// TIA Portal project "Tripping_hoya" (V16)

(* hardware
DEVICE "S7-1200 station_1"  S7-1200 Station
   slot 0: "Rack_0"  S7-1200 Rack  Rack  V1.0
   slot 1: "PLC_1"  CPU 1214C AC/DC/Rly  6ES7 214-1BG40-0XB0  V4.4
   slot 2: "DI 16x24VDC/DQ 16xRelay_1"  SM 1223 DI16/DQ16 x relay  6ES7 223-1PL32-0XB0  V2.0
   slot 3: "DI 16x24VDC/DQ 16xRelay_2"  SM 1223 DI16/DQ16 x relay  6ES7 223-1PL32-0XB0  V2.0
   slot 4: "DI 16x24VDC/DQ 16xRelay_3"  SM 1223 DI16/DQ16 x relay  6ES7 223-1PL32-0XB0  V2.0
   slot 5: "DQ 8x24VDC _1"  SM 1222 DQ8 x 24VDC  6ES7 222-1BF32-0XB0  V2.0
   slot 6: "DI 16x24VDC_1"  6ES7 221-1BH32-0XB0  V2.0
   slot 7: "DI 16x24VDC_2"  6ES7 221-1BH32-0XB0  V2.0
   slot 101: "CM 1241 (RS232)_1"  6ES7 241-1AH32-0XB0  V2.2
*)

// ===== PLC "PLC_1"  CPU 1214C AC/DC/Rly =====

VAR_GLOBAL   // PLC tag table "Default tag table"
   "Start" AT %I0.0 : Bool;   // Tín hiệu nhấn nút start
   "Stop" AT %I0.1 : Bool;   // Tín hiệu nhấn nút stop
   "Reset" AT %I0.2 : Bool;   // Tín hiệu nhấn nút Reset
   "EMG" AT %I0.3 : Bool;
   "SS Up XL Chốt" AT %I0.4 : Bool;
   "SS Down XL Chốt" AT %I0.5 : Bool;
   "SS Up XL Cửa Input" AT %I0.6 : Bool;
   "SS Down XL Cửa Input" AT %I0.7 : Bool;
   "SS Up XL Nâng Input" AT %I1.0 : Bool;
   "SS Down XL Nâng Input" AT %I1.1 : Bool;
   "SS Input Rack" AT %I1.2 : Bool;   // Cảm biến có rack trong Xylanh nâng input
   "SS Chốt Rack Input" AT %I1.3 : Bool;
   "SS Rack Input XL" AT %I1.4 : Bool;
   "SS Limit 1 Tranfer1" AT %I1.5 : Bool;
   "SS Limit 1 Tranfer2" AT %I2.1 : Bool;
   "SS Open XL Robot" AT %I2.3 : Bool;
   "SS Close XL Robot" AT %I2.4 : Bool;
   "SS Down XL Robot" AT %I2.5 : Bool;
   "SS Up XL Robot" AT %I2.6 : Bool;   // Cảm biến Xy Lanh dọc của Robot
   "SS XL Up Cửa Output" AT %I2.7 : Bool;
   "SS XL Down Cửa Output" AT %I3.0 : Bool;
   "SS Up XL Nâng Output" AT %I3.1 : Bool;
   "SS Down XL Nâng Output" AT %I3.2 : Bool;
   "SS Up XL Lift 1" AT %I5.5 : Bool;
   "SS Down XL Lift 1" AT %I5.6 : Bool;   // Trgger DOwnnXLn3
   "SS Up XL Lift 5" AT %I5.7 : Bool;
   "SS Down XL Lift 5" AT %I6.0 : Bool;
   "SS HW Tank1" AT %I6.1 : Bool;
   "SS LW Tank1" AT %I6.2 : Bool;
   "SS HW Tank2" AT %I6.3 : Bool;
   "SS LW Tank2" AT %I6.4 : Bool;
   "SS HW Tank3" AT %I6.5 : Bool;
   "SS LW Tank3" AT %I6.6 : Bool;
   "SS HW Tank4" AT %I6.7 : Bool;
   "SS LW Tank4" AT %I7.0 : Bool;
   "SS HW Tank5" AT %I7.1 : Bool;
   "SS LW Tank5" AT %I7.2 : Bool;
   "SS HW Tank6" AT %I7.3 : Bool;
   "SS LW Tank6" AT %I7.4 : Bool;
   "SS HW Tank7" AT %I7.5 : Bool;
   "SS LW Tank7" AT %I7.6 : Bool;
   "SS HW Tank8" AT %I7.7 : Bool;
   "SS LW Tank8" AT %I8.0 : Bool;
   "SS HW Tank9" AT %I8.1 : Bool;
   "SS LW Tank9" AT %I8.2 : Bool;
   "SS W Tank1" AT %I8.5 : Bool;
   "SS W Tank2" AT %I8.6 : Bool;
   "SS W Tank3" AT %I8.7 : Bool;
   "SS W Tank4" AT %I9.0 : Bool;
   "SS W Tank5" AT %I9.1 : Bool;
   "SS W Tank6" AT %I9.2 : Bool;
   "SS W Tank7" AT %I9.3 : Bool;
   "SS W Tank8" AT %I9.4 : Bool;
   "SS W Tank9" AT %I9.5 : Bool;
   "SS Rack BT Out" AT %I9.7 : Bool;
   "Up_Limit_Lift" AT %I10.2 : Bool;   // Cảm Biến Trên Axis Lift
   "Down_Limit_Lift" AT %I10.3 : Bool;   // Cảm biến Dưới Axis Lift
   "Jog + Robot" AT %I10.4 : Bool;   // Trigger JOG +
   "Jog - Robot" AT %I10.5 : Bool;   // Trigger JOG -
   "SS Up XL Lift 2" AT %I10.6 : Bool;   // Cảm Biến Trên Xy Lanh Nâng Bath 4
   "SS Down XL Lift 2" AT %I10.7 : Bool;   // Cảm Biến Dưới Xy Lanh Nâng Bath 4
   "SS Up XL Lift 3" AT %I11.0 : Bool;   // Cảm Biến Trên Xy Lanh Nâng Bath 5
   "SS Down XL Lift 3" AT %I11.1 : Bool;   // Cảm Biến Dưới Xy Lanh Nâng Bath 5
   "SS Up XL Lift 4" AT %I11.2 : Bool;   // Cảm Biến Trên Xy Lanh Nâng Bath 6
   "SS Down XL Lift 4" AT %I11.3 : Bool;   // Cảm Biến Dưới Xy Lanh Nâng Bath 6
   "SS_Cửa_Khung" AT %I11.4 : Bool;
   "Right_Limit_X" AT %I11.5 : Bool;
   "Left_Limit_X" AT %I11.6 : Bool;
   "XL Chốt Input_1" AT %Q0.0 : Bool;
   "XL Chốt Input_2" AT %Q0.1 : Bool;
   "XL Cửa Input_1" AT %Q0.2 : Bool;
   "XL Cửa Input_2" AT %Q0.3 : Bool;
   "XL Nâng Input1" AT %Q0.4 : Bool;
   "XL Nâng Input2" AT %Q0.5 : Bool;
   "XL Kẹp Robot_1" AT %Q0.6 : Bool;
   "XL Kẹp Robot_2" AT %Q0.7 : Bool;
   "Motor Băng tải Input" AT %Q1.0 : Bool;
   "XL Cửa Output_1" AT %Q1.1 : Bool;
   "XL Cửa Output_2" AT %Q2.0 : Bool;
   "XL Nâng Output1" AT %Q2.1 : Bool;
   "XL Nâng Output2" AT %Q2.2 : Bool;
   "Motor Băng Tải Output" AT %Q2.3 : Bool;
   "Van DI ON" AT %Q2.4 : Bool;
   "Van DI OFF" AT %Q2.5 : Bool;
   "Pump Bath1" AT %Q2.6 : Bool;
   "Pump Bath2" AT %Q2.7 : Bool;
   "Pump Bath3" AT %Q3.0 : Bool;
   "Pump Bath4" AT %Q3.1 : Bool;
   "Pump Bath5" AT %Q3.2 : Bool;
   "Pump Bath6" AT %Q3.3 : Bool;
   "Pump Bath7" AT %Q3.4 : Bool;
   "Pump Bath8" AT %Q3.5 : Bool;
   "Pump Bath9" AT %Q3.6 : Bool;
   "Pump Bath10" AT %Q3.7 : Bool;
   "Van RO ON" AT %Q4.0 : Bool;
   "Van RO OFF" AT %Q4.1 : Bool;
   "UltraS Tank1" AT %Q4.5 : Bool;
   "UltraS Tank2" AT %Q4.6 : Bool;
   "UltraS Tank3" AT %Q4.7 : Bool;
   "UltraS Tank4" AT %Q5.0 : Bool;
   "UltraS Tank5" AT %Q5.1 : Bool;
   "UltraS Tank6" AT %Q5.2 : Bool;
   "UltraS Tank7" AT %Q5.3 : Bool;
   "UltraS Tank8" AT %Q5.4 : Bool;
   "UltraS Tank9" AT %Q5.5 : Bool;
   "XL Lift 1_1" AT %Q6.0 : Bool;
   "XL Lift 1_2" AT %Q6.1 : Bool;
   "XL Lift 2_1" AT %Q6.2 : Bool;
   "XL Lift 2_2" AT %Q6.3 : Bool;
   "XL Lift 3_1" AT %Q6.4 : Bool;
   "XL Lift 3_2" AT %Q6.5 : Bool;
   "XL Lift 4_1" AT %Q6.6 : Bool;
   "XL Lift 4_2" AT %Q6.7 : Bool;
   "XL Lift 5_1" AT %Q7.0 : Bool;
   "XL Lift 5_2" AT %Q7.1 : Bool;
   "Red Lamp" AT %Q7.2 : Bool;
   "Yellow Lamp" AT %Q7.3 : Bool;
   "Green Lamp" AT %Q7.4 : Bool;
   "Buzzer" AT %Q7.5 : Bool;
   "XL_UP_Robot" AT %Q7.6 : Bool;
   "XL_DOWN_Robot" AT %Q7.7 : Bool;
   "System_Byte" AT %MB1 : Byte;
   "FirstScan" AT %M1.0 : Bool;
   "DiagStatusUpdate" AT %M1.1 : Bool;
   "AlwaysTRUE" AT %M1.2 : Bool;
   "AlwaysFALSE" AT %M1.3 : Bool;
   "Clock_Byte" AT %MB0 : Byte;
   "Clock_10Hz" AT %M0.0 : Bool;
   "Clock_5Hz" AT %M0.1 : Bool;
   "Clock_2.5Hz" AT %M0.2 : Bool;
   "Clock_2Hz" AT %M0.3 : Bool;
   "Clock_1.25Hz" AT %M0.4 : Bool;
   "Clock_1Hz" AT %M0.5 : Bool;
   "Clock_0.625Hz" AT %M0.6 : Bool;
   "Clock_0.5Hz" AT %M0.7 : Bool;
   "DISCONNECT_TCP_PC_TRGGER" AT %M2.0 : Bool;   // Tín hiệu ngắt kết nối từ PC
   "SEND_TCP_TRIGGER" AT %M2.1 : Bool;   // Tín Hiệu Gửi TCP 1
   "SEND_TCP_TRIGGER_1" AT %M2.2 : Bool;   // Tín Hiệu Gủi TCP 2
   "SEND_TCP_TRIGGER_2" AT %M2.3 : Bool;   // Tín Hiệu Gửi TCP 3
   "SEND_REQ" AT %M2.4 : Bool;   // Tín Hiệu Kích Gửi
   "length" AT %MW4 : Int;   // Biến Lưu Chiều Dài Data cần gửi
   "Edge_1" AT %M2.5 : Bool;   // Temp Pulse 1
   "Axis_x_Home" AT %M2.6 : Bool;   // Axis X Home trigger
   "Edge_2" AT %M2.7 : Bool;   // Temp Pulse 2
   "SYSTEM_READY" AT %M3.0 : Bool;   // READY STATUS
   "MANUAL_STATE" AT %M3.1 : Bool;   // Chế độ manual
   "AUTO_STATE" AT %M3.2 : Bool;   // Chế Dộ AUTO
   "HOME_MAN_TRIGGER_PC" AT %M3.3 : Bool;   // Tín Hiệu Home Manual
   "HOME_AUTO_TRIGGER_PC" AT %M3.4 : Bool;   // Tín HIệu HOME AUTO
   "SELECT_AXIS_HOME" AT %MW6 : Int;   // 0-ALL Axis , 1 - AXIS X, 2 - AXIS LIFT
   "Edge_3" AT %M3.5 : Bool;   // Temp Pulse 3
   "Edge_4" AT %M3.6 : Bool;   // Temp Pulse 4
   "Edge_5" AT %M3.7 : Bool;   // Temp 5
   "Edge_6" AT %M8.0 : Bool;   // Temp6
   "Edge_7" AT %M8.1 : Bool;   // Temp 7
   "Edge_8" AT %M8.2 : Bool;   // Temp 8
   "Edge_9" AT %M8.3 : Bool;   // Temp 9
   "Edge_10" AT %M8.4 : Bool;   // Temp 10
   "Move_Point_X" AT %M8.5 : Bool;   // Trigger_Move_Point Axis X
   "Edge_11" AT %M8.6 : Bool;   // Temp 11
   "Move_Point_LIFT" AT %M8.7 : Bool;   // Tín Hiệu Move Point Axis LIFT
   "WRITE_DATA_POINT_X" AT %M9.0 : Bool;   // Trigger Cài đặt điểm
   "Edge_12" AT %M9.1 : Bool;   // Temp 12
   "Edge_13" AT %M9.2 : Bool;   // Temp 13
   "WRITE_DATA_POINT_LIFT" AT %M9.3 : Bool;   // Trigger Set data point Axis LIft
   "Jog_TF_1_FW" AT %M9.4 : Bool;   // Trigger Jog FW Tranfer 1
   "Edge_14" AT %M9.5 : Bool;   // Temp 14
   "Edge_15" AT %M9.6 : Bool;   // Temp 15
   "Edge_16" AT %M9.7 : Bool;   // Temp 16
   "Edge_17" AT %M10.0 : Bool;   // Temp 17
   "Jog_TF_1_BW" AT %M10.1 : Bool;   // Trigger Jog BW Tranfer 1
   "Jog_TF_2_FW" AT %M10.2 : Bool;   // Trigger Jog FW Tranfer 2
   "Edge_18" AT %M10.3 : Bool;   // Temp 18
   "Edge_19" AT %M10.4 : Bool;   // Temp 19
   "Jog_TF_2_BW" AT %M10.5 : Bool;   // Trigger Jog BW Tranfer 2
   "Edge_20" AT %M10.6 : Bool;   // Temp 20
   "Edge_21" AT %M10.7 : Bool;   // Temp 21
   "Run_TF_1_FW" AT %M11.0 : Bool;   // Trgger Run FW Tranfer 1
   "Edge_22" AT %M11.1 : Bool;   // Temp 22
   "Edge_23" AT %M11.2 : Bool;   // Temp 23
   "Run_TF_1_BW" AT %M11.3 : Bool;   // Trgger Run BW Tranfer 1
   "Edge_24" AT %M11.4 : Bool;   // Temp 24
   "Edge_25" AT %M11.5 : Bool;   // Temp 25
   "Run_TF_2_FW" AT %M11.6 : Bool;   // Trigger Run FW Tranfer 2
   "Edge_26" AT %M11.7 : Bool;   // Temp 26
   "Edge_27" AT %M12.0 : Bool;   // Temp 27
   "Run_TF_2_BW" AT %M12.1 : Bool;   // Trigger Run BW Tranfer 2
   "Edge_28" AT %M12.2 : Bool;   // Temp 28
   "Edge_29" AT %M12.3 : Bool;   // Temp 29
   "Jog_Lift_1_FW" AT %M12.4 : Bool;   // Trigger Jog Lift 1 FW
   "Edge_30" AT %M12.5 : Bool;   // Temp 30
   "Edge_31" AT %M12.6 : Bool;   // Temp 31
   "Jog_Lift_1_BW" AT %M12.7 : Bool;   // Trgger Jog Lift 1 BW
   "Edge_32" AT %M13.0 : Bool;   // Temp 32
   "Edge_33" AT %M13.1 : Bool;   // Temp 33
   "Run_Lift_1_FW" AT %M13.2 : Bool;   // Trigger Run Lift 1 FW
   "Edge_34" AT %M13.3 : Bool;   // Temp 34
   "Edge_35" AT %M13.4 : Bool;   // Temp 35
   "Run_Lift_1_BW" AT %M13.5 : Bool;   // Trigger Run Lift 1 BW
   "Edge_36" AT %M13.6 : Bool;   // Temp 36
   "Edge_37" AT %M13.7 : Bool;   // Temp 37
   "Jog_Lift_2_FW" AT %M14.0 : Bool;   // Trigger Jog Lifft 2 FW
   "Edge_38" AT %M14.1 : Bool;   // Temp 38
   "Edge_39" AT %M14.2 : Bool;   // Temp 39
   "Jog_Lift_2_BW" AT %M14.3 : Bool;   // Trigger Jog Lift 2 BW
   "Edge_40" AT %M14.4 : Bool;   // Temp 40
   "Edge_41" AT %M14.5 : Bool;   // Temp 41
   "Run_Lift_2_FW" AT %M14.6 : Bool;   // Trigger Run Lift 2 FW
   "Edge_42" AT %M14.7 : Bool;   // Temp 42
   "Edge_43" AT %M15.0 : Bool;   // Temp 43
   "Run_Lift_2_BW" AT %M15.1 : Bool;   // Trigger Run Lifr 2 BW
   "Edge_44" AT %M15.2 : Bool;   // Temp 44
   "Edge_45" AT %M15.3 : Bool;   // Temp 45
   "Jog_Lift_3_FW" AT %M15.4 : Bool;   // Trgger Jog Lift 3 FW
   "Edge_46" AT %M15.5 : Bool;   // Temp 46
   "Edge_47" AT %M15.6 : Bool;   // Temp 47
   "Jog_Lift_3_BW" AT %M15.7 : Bool;   // Trigger Jog Lift 3 BW
   "Edge_48" AT %M16.0 : Bool;   // Temp 48
   "Edge_49" AT %M16.1 : Bool;   // Temp 49
   "Run_Lift_3_FW" AT %M16.2 : Bool;   // Trigger Run Lift 3 FW
   "Edge_50" AT %M16.3 : Bool;   // Temp 50
   "Edge_51" AT %M16.4 : Bool;   // Temp 51
   "Run_Lift_3_BW" AT %M16.5 : Bool;   // Trigger Run Lift 3 BW
   "Edge_52" AT %M16.6 : Bool;   // Temp 52
   "Edge_53" AT %M16.7 : Bool;   // Temp 53
   "SET_FREQ_MOTOR_TRANFER" AT %M17.0 : Bool;   // Tín hiệu set freq cho Motor tranfer
   "SET_ACC_DEC_MOTOR_TRANFER" AT %M17.1 : Bool;
   "Edge_54" AT %M17.2 : Bool;   // Temp 54
   "Edge_55" AT %M17.3 : Bool;   // Temp 55
   "SET_FREQ_MOTOR_LIFT" AT %M17.4 : Bool;   // Tín hiệu cài đặt tần số cho đọng cơ nhúng
   "Edge_56" AT %M17.5 : Bool;   // Temp 56
   "SET_ACC_DEC_MOTOR_LIFT" AT %M17.6 : Bool;   // Tín hiệu cài đặt thời gian tăng tốc giảm tốc của động cơ nhúng
   "Edge_57" AT %M17.7 : Bool;   // Temp 57
   "Man_Axis_X" AT %I8.3 : Bool;   // Biến Chọn Manual Axis X
   "Man_Axis_Lift" AT %I8.4 : Bool;   // Biến Chọn Manual Axis Lift
   "Begin_Reset" AT %M18.0 : Bool;   // Reset Trgger
   "Stop_Pump_temp_1" AT %M18.1 : Bool;
   "RESET_PUMP_1" AT %M18.2 : Bool;
   "START_PUMP_1" AT %M18.3 : Bool;
   "STOP_PUMP_1" AT %M18.4 : Bool;
   "Stop_Pump_temp_2" AT %M18.5 : Bool;
   "RESET_PUMP_2" AT %M18.6 : Bool;
   "START_PUMP_2" AT %M18.7 : Bool;
   "STOP_PUMP_2" AT %M19.0 : Bool;
   "Stop_Pump_temp_3" AT %M19.1 : Bool;
   "RESET_PUMP_3" AT %M19.2 : Bool;
   "START_PUMP_3" AT %M19.3 : Bool;
   "STOP_PUMP_3" AT %M19.4 : Bool;
   "Stop_Pump_temp_4" AT %M19.5 : Bool;
   "RESET_PUMP_4" AT %M19.6 : Bool;
   "START_PUMP_4" AT %M19.7 : Bool;
   "STOP_PUMP_4" AT %M20.0 : Bool;
   "Stop_Pump_temp_5" AT %M20.1 : Bool;
   "RESET_PUMP_5" AT %M20.2 : Bool;
   "START_PUMP_5" AT %M20.3 : Bool;
   "STOP_PUMP_5" AT %M20.4 : Bool;
   "Stop_Pump_temp_6" AT %M20.5 : Bool;
   "RESET_PUMP_6" AT %M20.6 : Bool;
   "START_PUMP_6" AT %M20.7 : Bool;
   "STOP_PUMP_6" AT %M21.0 : Bool;
   "Stop_Pump_temp_7" AT %M21.1 : Bool;
   "RESET_PUMP_7" AT %M21.2 : Bool;
   "START_PUMP_7" AT %M21.3 : Bool;
   "STOP_PUMP_7" AT %M21.4 : Bool;
   "Stop_Pump_temp_8" AT %M21.5 : Bool;
   "START_PUMP_8" AT %M21.6 : Bool;
   "RESET_PUMP_8" AT %M21.7 : Bool;
   "STOP_PUMP_8" AT %M22.0 : Bool;
   "Stop_Pump_temp_9" AT %M22.1 : Bool;
   "RESET_PUMP_9" AT %M22.2 : Bool;
   "STOP_PUMP_9" AT %M22.3 : Bool;
   "START_PUMP_9" AT %M22.4 : Bool;
   "Home_Tranfer" AT %M22.5 : Bool;   // Home Tranfer
   "Edge_58" AT %M22.6 : Bool;   // Temp 58
   "Initial_Tranfer" AT %M22.7 : Bool;   // Initail Tranfer Group
   "Stop_JOG_Tranfer" AT %M23.0 : Bool;   // Stop Signal Tranfer
   "Current_timer_Count" AT %MD24 : Time;   // Biến nhớ Time Hiện Tại
   "Prepare_BW_TF_1" AT %M23.1 : Bool;   // Signal backward tranfer group
   "Edge_59" AT %M23.2 : Bool;   // Temp 59
   "Edge_60" AT %M23.3 : Bool;   // Temp 60
   "BW_Tranfer" AT %M23.4 : Bool;   // Signal Trigger BW
   "Edge_61" AT %M23.5 : Bool;   // Temp 61
   "Up_XL_Lift_1" AT %M23.6 : Bool;   // Trigger Up Xy Lanh 1
   "Down_XL_Lift_1" AT %M23.7 : Bool;   // Trigger Down Xy Lạnh 1
   "Down_XL_Lift_2" AT %M28.0 : Bool;   // Trgger Down XL 2
   "Up_XL_Lift_2" AT %M28.1 : Bool;   // Trigger Up XL 2
   "Up_XL_Lift_3" AT %M28.2 : Bool;   // Trigger XL Lift 3
   "Down_XL_Lift_3" AT %M28.3 : Bool;   // Trigger Down XL Lift 3
   "Up_XL_Lift_4" AT %M28.4 : Bool;   // Trgger Up XL Lift 4
   "Down_XL_Lift_4" AT %M28.5 : Bool;   // Trgger Down XL Lift 4
   "Up_XL_Lift_5" AT %M28.6 : Bool;   // Trgger Up XL Lift 5
   "Down_XL_Lift_5" AT %M28.7 : Bool;   // Trigger Down XL 5
   "Manual_Up_XL_Lift_1" AT %M29.0 : Bool;   // Trigger Manual Up XL Lift 1
   "Manual_Down_XL_Lift_1" AT %M29.1 : Bool;   // Trigger manual Down XL Lift 1
   "Manual_Up_XL_Lift_2" AT %M29.2 : Bool;   // Trgger Manual Up XL Lift 2
   "Manual_Down_XL_Lift_2" AT %M29.3 : Bool;   // Trigger Manual Down XL Lift 2
   "Manual_Up_XL_Lift_3" AT %M29.4 : Bool;   // Trigger Manual Up XL Lift 3
   "Manual_Down_XL_Lift_3" AT %M29.5 : Bool;   // Trigger Manual Down XL Lift 3
   "Manual_Up_XL_Lift_4" AT %M29.6 : Bool;   // Trigger Manual Up XL Lift 4
   "Manual_Down_XL_Lift_4" AT %M29.7 : Bool;   // Trigger Manual Down XL Lift 4
   "Manual_Up_XL_Lift_5" AT %M30.0 : Bool;   // Trigger Manual Up XL Lift 5
   "Manual_Down_XL_Lift_5" AT %M30.1 : Bool;   // Trigger Manual Down XL Lift 5
   "Up_XL_Chốt" AT %M30.2 : Bool;   // Signal Up Xy Lanh Chốt
   "Manual_Up_XL_Chốt_Input" AT %M30.3 : Bool;   // Trigger manual Up Xy Lanh Chốt In put
   "Down_XL_Chốt" AT %M30.4 : Bool;   // Trigger Down Xy Lanh Chốt Input
   "Manual_Down_XL_Chốt_Input" AT %M30.5 : Bool;   // Trigger Manual Down Xy lanh CHót Input
   "Up_XL_Nâng Input" AT %M30.6 : Bool;   // Trigger Up XL nâng input
   "Manual_Up_XL_Nâng_Input" AT %M30.7 : Bool;   // Trigger manual up Xy lanh nâng input
   "Down_XL_Nâng Input" AT %M31.0 : Bool;   // Trigger Down XL Nâng input
   "Manual_Down_XL_Nâng_Input" AT %M31.1 : Bool;   // Trigger Manual Down XL nâng input
   "Up_XL_Nâng Output" AT %M31.2 : Bool;   // Trigger Up XL Nâng Input
   "Down_XL_Nâng Output" AT %M31.3 : Bool;   // Trigger Up XL Nâng Output
   "Manual_Down_XL_Nâng_ Output" AT %M31.4 : Bool;   // Trigger Manual Down XL Nâng Input
   "CLose_XL_Kẹp_Robot" AT %M31.5 : Bool;   // Trigger Close XL Kẹp Robot
   "Manual_Close_XL_Kẹp_Robot" AT %M31.6 : Bool;   // Trigger Manual Close Xl Kẹp Robot
   "Open_XL_Kẹp_Robot" AT %M31.7 : Bool;   // Trigger Open XL Kẹp Robot
   "Manual_Open_XL_Kẹp_Robot" AT %M32.0 : Bool;   // Trigger Manual Open XL Kẹp Robot
   "Up_XL_Robot" AT %M32.1 : Bool;   // Trigger Up XL Robot
   "Manual_Up_XL_Robot" AT %M32.2 : Bool;   // Trigger Manual Up XL Robot
   "Down_XL_Robot" AT %M32.3 : Bool;   // Trigger Down XL Robot
   "Manual_Down_XL_Robot" AT %M32.4 : Bool;   // Trigger Manual Down XL Robot
   "Edge_62" AT %M32.5 : Bool;   // Temp 62
   "No_rack" AT %M32.6 : Bool;   // Signal Detect Has Any Rack In Machine
   "TF1_Position_1" AT %M32.7 : Bool;   // Signal Detect TF1 at Position 1
   "Trigger_Run_FW_TF1" AT %M33.0 : Bool;   // Signal Run FW TF Excute
   "TF1_Position_2" AT %M33.1 : Bool;   // Signal Detect Tranfer 1 at Position 2
   "Stop_Run_FW_TF1" AT %M33.2 : Bool;   // Signal to Stop Run Forward Tranffer 1
   "Stop_Run_BW_TF1" AT %M33.3 : Bool;   // Signal to stop run backward Tranfer 1
   "Trigger_Run_BW_TF1" AT %M33.4 : Bool;   // Signal Run Backward Tranfer1
   "Being_TF1_FW" AT %M33.5 : Bool;   // Status FW of TF1
   "Being_TF1_BW" AT %M33.6 : Bool;   // Status BW of TF1
   "Mem_Status_1" AT %M33.7 : Bool;   // Memory 1
   "Begin_Tripping" AT %M34.0 : Bool;   // Signal To Tripping Area 1
   "Edge_63" AT %M34.1 : Bool;   // Temp 63
   "Down_XL_Lift_1_Excute" AT %M34.2 : Bool;   // Excute Down XL Lift 1
   "Edge_64" AT %M34.3 : Bool;   // Temp 64
   "Stop_Delay_Temp_1" AT %M34.4 : Bool;   // Mem temp 1
   "Tripping_Area1_Done" AT %M34.5 : Bool;   // Signal Detect Tripping Process Done
   "Up_XL_Lift_1_Excute" AT %M34.6 : Bool;   // Excute Up XL Liff 1
   "Trigger_Trip_Area1" AT %M34.7 : Bool;   // Trigger To Excute Begin Tranffer
   "Trigger_Trip_Area3" AT %M35.0 : Bool;   // Trigger to Excute Tripping process Area 3
   "TF2_Position_1" AT %M35.1 : Bool;   // Signal Detect TF2 at Possiontion 1
   "TF2_Position_2" AT %M35.2 : Bool;   // Signal Detect TF2 at Position 2
   "Stop_Run_FW_TF2" AT %M35.3 : Bool;   // Stop Signal Run TF2 FW
   "Trigger_Run_FW_TF2" AT %M35.4 : Bool;   // Trigger to Run FW TF2
   "Being_TF2_FW" AT %M35.5 : Bool;   // Status Run FW TF2
   "Stop_Run_BW_TF2" AT %M35.6 : Bool;   // Signal To Stop Run BW TF2
   "Trigger_Run_BW_TF2" AT %M35.7 : Bool;   // Trigger to Run BW TF2
   "Being_TF2_BW" AT %M36.0 : Bool;   // Status Run BW TF2
   "Down_XL_Lift_5_Excute" AT %M36.1 : Bool;   // Trigger Down XL 5 Excute
   "Mem_Status_2" AT %M36.2 : Bool;   // Memory temp 2
   "Begin_Tripping_1" AT %M36.3 : Bool;   // Signal To Tripping Area3
   "Stop_Delay_Temp_2" AT %M36.4 : Bool;   // Mem Temp 2
   "Edge_65" AT %M36.5 : Bool;   // Temp 65
   "Edge_66" AT %M36.6 : Bool;   // Temp 66
   "Up_XL_Lift_5_Excute" AT %M36.7 : Bool;   // Excute Up XL Lift 5
   "Back_To_Posiont1_TF1" AT %M37.0 : Bool;   // Signal to back to postion 1
   "Prepare_Stop_TF1" AT %M37.1 : Bool;   // Signal To prepare stop TF1
   "Descrease_Speed_TF1" AT %M37.2 : Bool;   // Signal To Descrease Speed Of Tranfer 1
   "Edge_67" AT %M37.3 : Bool;   // Temp 67
   "Edge_68" AT %M37.4 : Bool;   // Temp 68
   "Waiting_SS_off_1" AT %M37.5 : Bool;   // Biến đợi cảm biến tắt lần 1
   "Edge_69" AT %M37.6 : Bool;   // Temp 69
   "Jog_home_TF1_BW_Excute" AT %M37.7 : Bool;   // Trigger Jog BW TF1 (1)
   "Waiting_SS_on_1" AT %M38.0 : Bool;   // Biến Đợi Cảm Biến TF1 On
   "Edge_70" AT %M38.1 : Bool;   // Temp70
   "Edge_71" AT %M38.3 : Bool;   // Temp 71
   "Original_TF" AT %M38.4 : Bool;   // ON: Đã Về gốc Tranfer, OFF: Đang hoặc chưa được về gốc
   "Edge_72" AT %M38.5 : Bool;   // Temp 72
   "Edge_73" AT %M38.6 : Bool;   // Temp 73
   "Edge_74" AT %M38.7 : Bool;   // Temp 74
   "Stop_JOG_Tranfer_1" AT %M39.0 : Bool;
   "Back_To_Posiont1_TF2" AT %M39.1 : Bool;
   "Original_TF_2" AT %M39.2 : Bool;
   "Prepare_Stop_TF2" AT %M39.3 : Bool;
   "Edge_75" AT %M39.4 : Bool;   // Temp 75
   "Edge_76" AT %M39.5 : Bool;   // Temp 76
   "Jog_home_TF2_BW_Excute" AT %M39.6 : Bool;
   "Current_timer_Count_2" AT %MD40 : Time;
   "Prepare_BW_TF_2" AT %M39.7 : Bool;
   "Initial_Tranfer_2" AT %M44.0 : Bool;
   "Waiting_SS_off_3" AT %M44.1 : Bool;
   "Edge_77" AT %M44.2 : Bool;
   "Edge_78" AT %M44.3 : Bool;
   "Waiting_SS_on_3" AT %M44.4 : Bool;
   "Prepare_BW_TF_3" AT %M44.5 : Bool;
   "Edge_79" AT %M44.6 : Bool;
   "Waiting_SS_off_4" AT %M44.7 : Bool;
   "Edge_80" AT %M45.0 : Bool;
   "Tripping_Area3_Done" AT %M45.1 : Bool;
   "Move_Avoid" AT %M45.2 : Bool;   // Trigger move to avoid robot
   "Move_Avoid_Excute" AT %M45.3 : Bool;   // Biến thực thi tránh robot
   "Stop_Move_Avoid" AT %M45.4 : Bool;   // Trigger To stop Avoid
   "Move_back_after_avoid" AT %M45.5 : Bool;
   "Move_back_after_avoid_Excute" AT %M45.6 : Bool;
   "Stop_Move_Back_Avoid" AT %M45.7 : Bool;
   "Signal_Active_Robot" AT %M46.0 : Bool;   // Tín hiệu báo hiệu khỏi động robot cho quá trình vove rack
   "Edge_81" AT %M46.1 : Bool;   // Temp 81
   "Start_Grab_Robot" AT %M46.2 : Bool;
   "Pick_From4_to_6" AT %M46.3 : Bool;   // Tín hiều di chuyển Rack từ Bath 4 đến Bath6
   "Pick_From4_to_5" AT %M46.4 : Bool;   // Tin hiệu di chuyển Rack dến Bath 5
   "At_Bath4" AT %M46.5 : Bool;   // Tín hiệu CHo biết Rack sẽ được nhúng ở Bath 4
   "Re_Signal_Start_Grab_Robot" AT %M46.6 : Bool;   // Tín hiệu gọi lại CỤm Robot
   "Move_Preocess_Robot_Excute" AT %M46.7 : Bool;   // Biến Khởi Động Chu trình Robot
   "Edge_82" AT %M47.0 : Bool;   // Temp 82
   "Robot_Move_P1_Started" AT %M47.1 : Bool;
   "Grabed_Rack" AT %M47.2 : Bool;   // Tín Hiệu báo hiệu đã kẹp rack
   "Pick_P1_Done" AT %M47.3 : Bool;   // Pick At P1 Robot Done
   "Edge_83" AT %M47.4 : Bool;   // Temp 83
   "Robot_Move_P2_Started" AT %M47.5 : Bool;
   "Edge_84" AT %M47.6 : Bool;   // Temp 84
   "Down_XL_Robot_1" AT %M47.7 : Bool;
   "Open_XL_Kẹp_Robot_1" AT %M48.0 : Bool;
   "Put_Rack_to_Bath" AT %M48.1 : Bool;
   "Up_XL_Robot_1" AT %M48.2 : Bool;
   "Put_Rack_Done" AT %M48.3 : Bool;
   "Edge_85" AT %M48.4 : Bool;   // Temp 85
   "Down_XL_Lift_Trgger" AT %M48.5 : Bool;
   "Down_XL_Lift_2_1" AT %M48.6 : Bool;
   "Down_XL_Lift_3_1" AT %M48.7 : Bool;
   "Down_XL_Lift_4_1" AT %M49.0 : Bool;
   "Manual_Jog + Robot" AT %M49.1 : Bool;   // Biến Manual Jog
   "Manual_Jog - Robot" AT %M49.2 : Bool;
   "Axis_X_Selection" AT %I3.3 : Bool;
   "Axis_Lift_Selection" AT %I3.4 : Bool;
   "Manual_Jog + Lift" AT %M49.3 : Bool;
   "Manual_Jog - Lift" AT %M49.4 : Bool;
   "Enable_Robot" AT %M49.5 : Bool;
   "Edge_86" AT %M49.6 : Bool;   // Temp 86
   "Disable_Robot" AT %M49.7 : Bool;
   "Edge_87" AT %M50.0 : Bool;   // Temp87
   "Enable_Lift" AT %M50.1 : Bool;
   "Edge_88" AT %M50.2 : Bool;   // Temp 88
   "Disable_Lift" AT %M50.3 : Bool;
   "Edge_89" AT %M50.4 : Bool;   // Temp 89
   "Manual_Jog_FW_TF1" AT %M50.5 : Bool;
   "Edge_90" AT %M50.6 : Bool;   // Temp 90
   "Edge_91" AT %M50.7 : Bool;   // Temp 91
   "Manual_Jog_BW_TF1" AT %M51.0 : Bool;
   "Edge_92" AT %M51.1 : Bool;
   "Edge_93" AT %M51.2 : Bool;
   "Manual_Jog_FW_TF2" AT %M51.3 : Bool;
   "Manual_Jog_BW_TF2" AT %M51.4 : Bool;
   "Edge_94" AT %M51.5 : Bool;   // Temp 94
   "Edge_95" AT %M51.6 : Bool;   // Temp96
   "Edge_96" AT %M51.7 : Bool;   // Temp 96
   "Edge_97" AT %M52.0 : Bool;   // Temp 97
   "Manual_Jog_FW_Lift1" AT %M52.1 : Bool;
   "Manual_Jog_BW_Lift1" AT %M52.2 : Bool;
   "Edge_98" AT %M52.3 : Bool;
   "Edge_99" AT %M52.4 : Bool;
   "Edge_100" AT %M52.5 : Bool;
   "Edge_101" AT %M52.6 : Bool;
   "Manual_Jog_FW_Lift2" AT %M52.7 : Bool;
   "Manual_Jog_BW_Lift2" AT %M53.0 : Bool;
   "Edge_102" AT %M53.1 : Bool;
   "Edge_103" AT %M53.2 : Bool;
   "Edge_104" AT %M53.3 : Bool;
   "Edge_105" AT %M53.4 : Bool;
   "Manual_Jog_FW_Lift3" AT %M53.5 : Bool;
   "Manual_Jog_BW_Lift3" AT %M53.6 : Bool;
   "Edge_106" AT %M53.7 : Bool;
   "Edge_107" AT %M54.0 : Bool;
   "Edge_108" AT %M54.1 : Bool;
   "Edge_109" AT %M54.2 : Bool;
   "Edge_110" AT %M54.3 : Bool;   // temp 110
   "Edge_111" AT %M54.4 : Bool;   // Temp 111
   "Edge_112" AT %M54.5 : Bool;   // Temp 112
   "Edge_113" AT %M54.6 : Bool;   // Temp 113
   "Manual_Run_FW_TF2" AT %M54.7 : Bool;
   "Manual_Run_BW_TF2" AT %M55.0 : Bool;
   "Manual_RUN_FW_Lift1" AT %M55.1 : Bool;
   "Manual_RUN_BW_Lift1" AT %M55.2 : Bool;
   "Edge_114" AT %M55.3 : Bool;
   "Edge_115" AT %M55.4 : Bool;
   "Edge_116" AT %M55.5 : Bool;
   "Edge_117" AT %M55.6 : Bool;
   "Manual_RUN_FW_Lift2" AT %M55.7 : Bool;
   "Manual_RUN_BW_Lift2" AT %M56.0 : Bool;
   "Edge_118" AT %M56.1 : Bool;
   "Edge_119" AT %M56.2 : Bool;
   "Edge_120" AT %M56.3 : Bool;
   "Edge_121" AT %M56.4 : Bool;
   "Manual_RUN_FW_Lift3" AT %M56.5 : Bool;
   "Manual_RUN_BW_Lift3" AT %M56.6 : Bool;
   "Edge_122" AT %M56.7 : Bool;
   "Edge_123" AT %M57.0 : Bool;
   "Edge_124" AT %M57.1 : Bool;
   "Edge_125" AT %M57.2 : Bool;
   "Manual_Run_FW_TF1" AT %M57.3 : Bool;
   "Manual_Run_BW_TF1" AT %M57.4 : Bool;
   "Edge_126" AT %M57.5 : Bool;
   "Edge_127" AT %M57.6 : Bool;
   "Edge_128" AT %M57.7 : Bool;
   "Edge_129" AT %M58.0 : Bool;
   "Brake_Lift" AT %Q4.2 : Bool;
   "Brake_Disable" AT %M58.1 : Bool;
   "Pump_9_On" AT %M58.2 : Bool;
   "Man_pump_9_on" AT %M58.3 : Bool;
   "Edge_130" AT %M58.4 : Bool;   // Temp 130
   "Edge_131" AT %M58.5 : Bool;   // Temp 131
   "Edge_132" AT %M58.6 : Bool;   // Temp 132
   "Pump_8_On" AT %M58.7 : Bool;
   "Man_pump_8_on" AT %M59.0 : Bool;
   "Pump_7_On" AT %M59.1 : Bool;
   "Man_pump_7_on" AT %M59.2 : Bool;
   "Pump_6_On" AT %M59.3 : Bool;
   "Man_pump_6_on" AT %M59.4 : Bool;
   "Pump_5_On" AT %M59.5 : Bool;
   "Man_pump_5_on" AT %M59.6 : Bool;
   "Pump_4_On" AT %M59.7 : Bool;
   "Man_pump_4_on" AT %M60.0 : Bool;
   "Pump_3_On" AT %M60.1 : Bool;
   "Man_pump_3_on" AT %M60.2 : Bool;
   "Pump_2_On" AT %M60.3 : Bool;
   "Man_pump_2_on" AT %M60.4 : Bool;
   "Pump_1_On" AT %M60.5 : Bool;
   "Man_pump_1_on" AT %M60.6 : Bool;
   "Edge_133" AT %M60.7 : Bool;   // Temp 133
   "PC_Kich_Have_Rack" AT %M61.0 : Bool;   // Pc Trigger has rack
   "Pressed" AT %M61.1 : Bool;
   "Edge_134" AT %M61.2 : Bool;   // Temp 134
   "Start_process" AT %M61.3 : Bool;
   "Test_" AT %M61.4 : Bool;
   "On_Robot" AT %M61.5 : Bool;
   "Auto_ON_Robot" AT %M61.6 : Bool;
   "Off_Robot" AT %M61.7 : Bool;
   "Auto_Off_Robot" AT %M62.0 : Bool;
   "On_Lift" AT %M62.1 : Bool;
   "Auto_ON_Lift" AT %M62.2 : Bool;
   "Off_Lift" AT %M62.3 : Bool;
   "Auto_Off_Lift" AT %M62.4 : Bool;
   "Lift_Rack_Up" AT %M62.5 : Bool;   // Kich Servo Lift Rack Up
   "Edge_135" AT %M62.6 : Bool;
   "Lift_Rack_Down" AT %M62.7 : Bool;
   "Edge_136" AT %M63.0 : Bool;
   "Move_Lift_to_PStart" AT %M63.1 : Bool;
   "Edge_137" AT %M63.2 : Bool;
   "Manual_Home_X" AT %M63.3 : Bool;
   "Edge_138" AT %M63.4 : Bool;
   "Auto_Home_X" AT %M63.5 : Bool;
   "Edge_139" AT %M63.6 : Bool;
   "Manual_Home_Lift" AT %M63.7 : Bool;
   "Auto_Home_Lift" AT %M64.0 : Bool;
   "Pause_Process" AT %M64.1 : Bool;
   "Up_XL_Lift_1_Init" AT %M64.2 : Bool;
   "Up_XL_Lift_2_Init" AT %M64.3 : Bool;
   "Up_XL_Lift_3_Init" AT %M64.4 : Bool;
   "Up_XL_Lift_4_Init" AT %M64.5 : Bool;
   "Up_XL_Lift_5_Init" AT %M64.6 : Bool;
   "Down_XL_Nâng Input_Init" AT %M64.7 : Bool;
   "Move_From5_to_6" AT %M65.0 : Bool;
   "Begin_Trip_Area_Robot" AT %M65.1 : Bool;
   "Req_For_Avoid" AT %M65.2 : Bool;
   "Temp_Time1" AT %MD66 : Time;
   "Temp_Time2" AT %MD70 : Time;
   "Tripping_Area_Robot_Done" AT %M65.3 : Bool;
   "Temp_Time_3" AT %MD74 : Time;
   "Up_XL_Lift_2_Robot_Trip_Done" AT %M65.4 : Bool;
   "Up_XL_Lift_3_Robot_Trip_Done" AT %M65.5 : Bool;
   "Up_XL_Lift_4_Robot_Trip_Done" AT %M65.6 : Bool;
   "Temp_Time_4" AT %MD78 : Time;
   "Move_From4_to_6" AT %M65.7 : Bool;
   "Not_Ready" AT %M82.0 : Bool;
   "Temp_Time5" AT %MD84 : Time;
   "Temp_Time_5" AT %MD88 : Time;
   "Temp_Time_6" AT %MD92 : Time;
   "Start_Grab_Robot_1" AT %M82.1 : Bool;
   "Edge_140" AT %M82.2 : Bool;
   "Waiting_for_Move_Robot" AT %M82.3 : Bool;
   "Edge_141" AT %M82.4 : Bool;
   "Step_1_Move_Done" AT %M82.5 : Bool;
   "Step_1_Move_Rack" AT %M82.6 : Bool;
   "Step_2_Move_Rack" AT %M82.7 : Bool;
   "Step_2_Move_Done" AT %M83.0 : Bool;
   "Press_Input_Rack" AT %M83.1 : Bool;
   "Motor Băng tải Input_2" AT %Q4.3 : Bool;
   "Run_FW_Conveyor_Input" AT %M83.2 : Bool;
   "Run_BW_Conveyor_Input" AT %M83.3 : Bool;
   "Run_Conveyor_Output" AT %M83.4 : Bool;
   "Stop_RunFW_Conveyor_Input" AT %M83.5 : Bool;
   "Run_CW_In" AT %M83.6 : Bool;
   "Stop_RunBW_Conveyor_Input" AT %M83.7 : Bool;
   "Waiting_To_Conveyor_Back" AT %M96.0 : Bool;
   "Stop_Wait_Temp" AT %M96.1 : Bool;
   "Up_XL_Nâng Output_Init" AT %M96.2 : Bool;
   "Wait_Lift_Input_Down" AT %M96.3 : Bool;
   "Wait_To_Confirm_Down_input" AT %M96.4 : Bool;
   "Stop_Wait_Confirm_Input" AT %M96.5 : Bool;
   "Check_Exist_Rack" AT %M96.6 : Bool;
   "Wait_To_Have_Rack" AT %M96.7 : Bool;
   "Stop_Wait_Have_Rack" AT %M97.0 : Bool;
   "Enable_Robot_Manual" AT %M97.1 : Bool;
   "Edge_142" AT %M97.2 : Bool;
   "Disable_Robot_Manual" AT %M97.3 : Bool;
   "Edge_143" AT %M97.4 : Bool;
   "Enable_Lift_Manual" AT %M97.5 : Bool;
   "Edge_144" AT %M97.6 : Bool;
   "Disable_Lift_Manual" AT %M97.7 : Bool;
   "Edge_145" AT %M98.0 : Bool;
   "Manual_Run_FW_Input_Conveyor" AT %M98.1 : Bool;
   "Manual_Run_BW_Input_Conveyor" AT %M98.2 : Bool;
   "Manual_RunFW_Output_Conveyor" AT %M98.3 : Bool;
   "ERROR_STATE" AT %M98.4 : Bool;
   "STOP_STATE" AT %M98.5 : Bool;
   "FIXED_ERROR" AT %M98.6 : Bool;
   "SS Limit 2 Tranfer1" AT %I2.0 : Bool;
   "SS Limit 2 Tranfer2" AT %I2.2 : Bool;
   "SS Limit 3 Tranfer2" AT %I3.5 : Bool;
   "Edge_146" AT %M38.2 : Bool;
   "Invalid_Vector" AT %M98.7 : Bool;
   "Invalid_Vector_1" AT %M99.0 : Bool;
   "Edge_147" AT %M99.1 : Bool;
   "Finish_Home_TF1" AT %M99.2 : Bool;
   "Finish_Home_TF1_1" AT %M99.3 : Bool;
   "Edge_148" AT %M99.4 : Bool;
   "Edge_149" AT %M99.5 : Bool;
   "Original_TF_1" AT %M99.6 : Bool;
   "Manual_Read_Data_Tranfer" AT %M99.7 : Bool;
   "Edge_150" AT %M100.0 : Bool;
   "Edge_151" AT %M100.1 : Bool;
   "Edge_152" AT %M100.2 : Bool;
   "Edge_153" AT %M100.3 : Bool;
   "Edge_154" AT %M100.4 : Bool;
   "Edge_155" AT %M100.5 : Bool;
   "Invalid_2_Vector" AT %M100.6 : Bool;
   "Invalid_2_Vector_1" AT %M100.7 : Bool;
   "Finish_Home_TF2" AT %M101.0 : Bool;
   "Finish_Home_TF2_1" AT %M101.1 : Bool;
   "Edge_156" AT %M101.2 : Bool;
   "Edge_157" AT %M101.3 : Bool;
   "EMG_TF" AT %M101.4 : Bool;
   "Manual_Home_TF1" AT %M101.5 : Bool;
   "Manual_Home_TF2" AT %M101.6 : Bool;
   "Edge_158" AT %M101.7 : Bool;
   "Edge_159" AT %M102.0 : Bool;
   "Edge_160" AT %M102.1 : Bool;
   "Edge_161" AT %M102.2 : Bool;
   "TF2_Position_3" AT %M102.3 : Bool;
   "Edge_162" AT %M102.4 : Bool;
   "EMG_SERVO_X" AT %M102.5 : Bool;
   "Edge_163" AT %M102.6 : Bool;
   "EMG_SERVO_LIFT" AT %M102.7 : Bool;
   "Manual_Up_XL_Nâng_Output" AT %M103.0 : Bool;
   "Manual_Up_XL_Nâng_Output(1)" AT %M103.1 : Bool;
   "Manual_Up_XL_Nâng_Output(2)" AT %M103.2 : Bool;
   "Open_VanDI" AT %M103.3 : Bool;
   "Manual_On_DI" AT %M103.4 : Bool;
   "Close_VanDI" AT %M103.5 : Bool;
   "Manual_Off_DI" AT %M103.6 : Bool;
   "Open_VanRO" AT %M103.7 : Bool;
   "Manual_On_RO" AT %M104.0 : Bool;
   "Close_VanRO" AT %M104.1 : Bool;
   "Manual_Off_RO" AT %M104.2 : Bool;
   "Test_ss" AT %M104.3 : Bool;
   "tess" AT %M104.4 : Bool;
   "Temp_Run_TF2_FW" AT %M104.5 : Bool;
   "Temp_Run_TF2_BW" AT %M104.6 : Bool;
   "Temp_Run_TF2_FW_1" AT %M104.7 : Bool;
   "Temp_Run_TF2_BW_1" AT %M105.0 : Bool;
   "Temp_Run_TF1_BW" AT %M105.1 : Bool;
   "Temp_Run_TF1_BW_1" AT %M105.2 : Bool;
   "Temp_Run_TF1_FW" AT %M105.3 : Bool;
   "Temp_Run_TF1_FW_1" AT %M105.4 : Bool;
   "Edge_164" AT %M105.5 : Bool;
   "Edge_165" AT %M105.6 : Bool;
   "Edge_166" AT %M105.7 : Bool;
   "Read_val" AT %MD106 : Real;
   "Flow_1" AT %IW64 : Word;
   "OUT_SCALE" AT %MD110 : Real;
   "Flow_Value_1" AT %MW114 : UInt;
   "Flow_2" AT %IW66 : Word;
   "Flow_Value_2" AT %MW116 : UInt;
   "Read_val_1" AT %MD118 : Real;
   "OUT_SCALE_1" AT %MD122 : Real;
   "Resume" AT %M126.0 : Bool;
   "Current_Position_X" AT %MW128 : Int;
   "Current_Position_Lift" AT %MW130 : Int;
   "Sync_Position" AT %M126.1 : Bool;
   "Trigger_Run_Convey_Out" AT %M126.2 : Bool;
   "New_Cycle_Trigger" AT %M126.3 : Bool;
   "Edge_167" AT %M126.4 : Bool;
   "Begin_Trip_A3" AT %M126.5 : Bool;
   "Begin_Trip_A1" AT %M126.6 : Bool;
   "Begin_Trip_All" AT %M126.7 : Bool;
   "Check_Tranfer_At_P1" AT %M127.0 : Bool;
   "Stop_Check_Tranfer" AT %M127.1 : Bool;
   "Edge_168" AT %M127.2 : Bool;
   "Edge_169" AT %M127.3 : Bool;
END_VAR

TYPE "Master_MB"
   STRUCT
      Req : Bool;
      MbAddress : Int := 1;
      Mode : USInt;
      DataAddr : UDInt;
      DataLen : UInt := 1;
      Done : Bool;
      Busy : Bool;
      Error : Bool;
      Status : Word;
      ErrorStatus : Word;
   END_STRUCT;
END_TYPE

TYPE "Type_MBLoad"
   STRUCT
      Done : Bool;
      Error : Bool;
      Status : Word;
      ErrorStatus : Word;
      DoneStored : Bool;
   END_STRUCT;
END_TYPE

TYPE "MasterData"
   STRUCT
      DataPtr : Array[0..8] of Int;
      SendData : Array[0..8] of Int;
      ReceivedData : Array[0..8] of Int;
      Status : Int;
      Array_Status : Array[0..15] of Bool;
      Current_Position : Array[0..1] of Int;
      Current_Speed : Array[0..1] of Int;
      ID : Int := 1;
      Current_Table_Point : Array[0..1] of Int;
      Select_Point : Int;
      Point_data : Int;
      Point_Speed : Int;
      "Point Accel" : Int := 50;
      "Point Decel" : Int := 50;
   END_STRUCT;
   // // Current_Table_Point[0] : Point Demand Value
   // // Current_Table_Point[1] : Point Actual Value
END_TYPE

TYPE "Process"
   STRUCT
      "Step" : USInt;
      Edge : Bool;
      mobusCommload : "Type_MBLoad";
      mobusMaster : "Master_MB";
      SingleDataAddr : Int;
      SingleDataLen : Int;
      SinggleData : Array[0..8] of Int;
      Write_Full_Done : Bool;
      SinggleMbAddr : UInt := 1;
      Step_W : UInt;
      Step_R : UInt;
   END_STRUCT;
END_TYPE

TYPE "Barcode"
   STRUCT
      Barcode_P1 : String[10];
      Barcode_P2 : String[1];
   END_STRUCT;
END_TYPE

TYPE "Barcode_pos"
   STRUCT
      Infor : "Barcode";
      Position : Int;
   END_STRUCT;
END_TYPE

DATA_BLOCK "SETTING_DATA"   // DB2
{ S7_Optimized_Access := 'FALSE' }
VERSION : 0.1
   VAR
      Point_to_Set : Int := 1;
      Point_Data : Int;
      "Point _Speed" : Int;
      Point_Accel : Int := 50;
      Point_Decel : Int := 50;
      Axis_Number : Int := 1;
   END_VAR
BEGIN
END_DATA_BLOCK

DATA_BLOCK "LIST_CODE_CHAR"   // DB3
{ S7_Optimized_Access := 'FALSE' }
VERSION : 0.1
   VAR
      Barcode_1 : "Barcode";   // Hàng Đợi Barcode 1
      Barcode_2 : "Barcode";   // Hàng Đợi Barcode 2
      Barcode_3 : "Barcode";   // Hàng Đợi Barcode 3
      Barcode_4 : "Barcode";   // Hàng Đợi Barcode 4
      Barcode_5 : "Barcode";   // Hàng Đợi Barcode 5
      Barcode_6 : "Barcode";   // Hàng Đợi Barcode 6
      Barcode_7 : "Barcode";   // Hàng Đợi Barcode 7
      Barcode_8 : "Barcode";   // Hàng Đợi Barcode 8
      Barcode_9 : "Barcode";   // Hàng Đợi Barcode 9
      Barcode_10 : "Barcode";   // Hàng Đợi Barcode 10
      Contain_In_Bath1 : "Barcode";
      Contain_In_Bath2 : "Barcode";
      Contain_In_Bath3 : "Barcode";
      Contain_In_Bath4 : "Barcode";
      Contain_In_Bath5 : "Barcode";
      Contain_In_Bath6 : "Barcode";
      Contain_In_Bath7 : "Barcode";
      Contain_In_Bath8 : "Barcode";
      Contain_In_Bath9 : "Barcode";
      Contain_In_Bath10 : "Barcode";
      Contain_In_Bath11 : "Barcode";
      Barcode_Queue_Robot : "Barcode";
   END_VAR
BEGIN
END_DATA_BLOCK

DATA_BLOCK "PROCESS_DATA_PARAMETER"   // DB5
{ S7_Optimized_Access := 'FALSE' }
VERSION : 0.1
   VAR
      Timer_Region1vs3 : Time := T#6m;
      Timer_Bath6_P1 : Time := T#6m;
      Timer_Bath6_P2 : Time := T#5m;
      Timer_Bath6_P3 : Time := T#3.5m;
      Timer_Bath6_P4 : Time := T#30s;
      Timer_Bath4_P2 : Time := T#5m;
      Timer_Bath4_P3 : Time := T#2m;
      Timer_Bath5_P4 : Time := T#5m;
      Tranfer_timer : Time := T#30s;
      Timer_temp_Robot_Area : Time;
      Current_TValue_Bath4 : Time;
      Current_TValue_Bath5 : Time;
      Current_TValue_Bath6 : Time;
      Current_TValue_Area_1 : Time;
      Current_TValue_Area_3 : Time;
      CurrentBathNumber : Int;   // Xác định vị trí bath có Rack được đưa vào { 1: Bath4, 2: Bath5, 3: Bath6}
      MODE : Int;   // 1: Manual, 0:Auto
      "Time_Int Check Sensor TF" : Int := 2000;
      "Time Check Sensor TF" : Time;
      Time_To_Active_Robot : Time := T#3s;
      Timer_Run_Conveyor_Inpur : Time := T#10s;
   END_VAR
BEGIN
END_DATA_BLOCK

DATA_BLOCK "RUN_TIME_PARAM"   // DB6
{ S7_Optimized_Access := 'FALSE' }
VERSION : 0.1
   VAR
      REQUEST_PICK_TYPE : Int;   // Biến xác định loại lỗi để Robot nhận biết để di chuyển đến các Bath phù hợp { 1: 4->6 ; 2:4->5; 3: 4->B4}
      VECTOR_ROBOT_MOVE : Array[0..1] of Int;
      CURRENT_BATH_DIP_ROBOT : Int;
      Current_TF1 : Int;
      Current_TF2 : Int;
      Current_Lift1 : Int;
      Current_Lift2 : Int;
      Current_Lift3 : Int;
   END_VAR
BEGIN
   // VECTOR_ROBOT_MOVE[0] : ĐIểm Đến Gắp (Bath4) || Bath5
   // VECTOR_ROBOT_MOVE[1] : Điểm Đến Thả (3: Bath5; 4: Bath6)
END_DATA_BLOCK

DATA_BLOCK "SYSTEM_DATA_RETAIN"   // DB10
{ S7_Optimized_Access := 'FALSE' }
VERSION : 0.1
   VAR
      Balance_temperature : Real := 60.0;
      Time_Wait_Down_XL_Lift_1 : Time := T#1S;
      Time_Wait_Down_XL_Lift_2 : Time := T#1S;
      Time_Wait_Down_XL_Lift_3 : Time := T#1S;
      Time_Wait_Down_XL_Lift_4 : Time := T#1S;
      Time_Wait_Down_XL_Lift_5 : Time := T#1S;
      TIme_Wait_Back_TF : Time := T#1S;   // Thời gian delay để tranfer quay về vị trí ban đầu
      Time_Wati_Move_RackB4 : Time := T#5S;
      Tranfer_Frequency : Real := 100.0;   // Tần số chạy Tranfer
      Dip_Frequency : Real := 50.0;
      Accel_Tranfer : Real := 0.5;
      Decel_Tranfer : Real := 0.5;
      Accel_Dip : Real := 0.5;
      Decel_Dip : Real := 0.5;
      BaudRate : UDInt := 57600;
      Parity : UDInt := 2;   // 0 - None; 1 - Odd; 2 - Even
      Detect_Vevtor : Int;
      Detect_Vevtor_1 : Int;
   END_VAR
BEGIN
END_DATA_BLOCK

DATA_BLOCK "Axis_X"   // DB12
{ S7_Optimized_Access := 'TRUE' }
VERSION : 0.1
// stored: InstanceOfName MB_Axis
"MB_Axis"
BEGIN
   Process.mobusMaster.MbAddress := 8;
   MasterData.ID := 8;
END_DATA_BLOCK

DATA_BLOCK "Axis_Lift"   // DB13
{ S7_Optimized_Access := 'TRUE' }
VERSION : 0.1
// stored: InstanceOfName MB_Axis
"MB_Axis"
BEGIN
   MasterData.ID := 2;
END_DATA_BLOCK

DATA_BLOCK "ROBOT_PARAM"   // DB14
{ S7_Optimized_Access := 'FALSE' }
VERSION : 0.1
   VAR
      JOG_X_SPEED : Int := 200;   // Tóc Độ jog X
      JOG_LIFT_SPEED : Int := 200;   // Tốc Độ Jog Y
      AxisRobot_Position_1 : Int;   // Tọa độ Bath4
      AxisRobot_Position_2 : Int;   // Tọa độ Bath5
      AxisRobot_Position_3 : Int;   // Tọa đồ Bath6
      AxisRobot_Position_Start : Int;   // Tọa độ Bắt Đầu Axis X
      AxisRobot_P1_Index : Int := 2;   // Chỉ mục bảng điểm Bath4
      AxisRobot_P2_Index : Int := 3;   // Chỉ mục Bảng điểm Bath 5
      AxisRobot_P3_Index : Int := 4;   // Chỉ mục Bảng điểm Bath6
      AxisRobot_PStart_Index : Int := 1;   // Chỉ mục bảng điểm Vị trí Bắt đầu
      AxisLift_Position_1 : Int := 0;   // Tọa Độ Lift Up
      AxisLift_Position_2 : Int := 0;   // Tọa Độ Lift Down
      AxisLift_Position_Start : Int := 0;   // Tọa Độ Bắt đầu Axis Lift
      AxisLift_P1_Index : Int := 2;   // Chỉ mục bảng điểm Lift Up
      AxisLift_P2_Index : Int := 3;   // Chỉ mục bảng ddierm Lift Down
      AxisLift_PStart_Index : Int := 1;   // Chỉ mục bảng điểm vị trí bắt đầu
      AxisRobot_Target_Point : Int := 1;   // Điểm đích cần đi chuyển đến
      AxisLift_Target_Point : Int := 1;   // Điểm đích cần đi chuyển đến
   END_VAR
BEGIN
END_DATA_BLOCK

DATA_BLOCK "Tranfer_1"   // DB15
{ S7_Optimized_Access := 'TRUE' }
VERSION : 0.1
// stored: InstanceOfName Inventer_Control
"Inventer_Control"
BEGIN
END_DATA_BLOCK

DATA_BLOCK "LIFT_1"   // DB16
{ S7_Optimized_Access := 'TRUE' }
VERSION : 0.1
// stored: InstanceOfName Inventer_Control
"Inventer_Control"
BEGIN
   ID := 4;
END_DATA_BLOCK

DATA_BLOCK "TCP_PARAMETER"   // DB17
{ S7_Optimized_Access := 'FALSE' }
VERSION : 0.1
   VAR
      REQ : Bool;
      DONE : Bool;
      BUSY : Bool;
      ERROR : Bool;
      STATUS : Word;
      DISCONNECT_REQ : Bool;
      DISCONNECT_DONE : Bool;
      DISCONNECT_ERROR : Bool;
      DISCONNECT_BUSY : Bool;
      DISCONNECT_STATUS : Word;
      SEND_REQ : Bool;
      DATA_LEN : Int;
      DATA : String;
      SEND_DONE : Bool;
      SEND_BUSY : Bool;
      SEND_ERROR : Bool;
      SEND_STATUS : Word;
   END_VAR
BEGIN
END_DATA_BLOCK

DATA_BLOCK "LIFT_2"   // DB18
{ S7_Optimized_Access := 'TRUE' }
VERSION : 0.1
// stored: InstanceOfName Inventer_Control
"Inventer_Control"
BEGIN
   ID := 5;
END_DATA_BLOCK

DATA_BLOCK "LIFT_3"   // DB19
{ S7_Optimized_Access := 'TRUE' }
VERSION : 0.1
// stored: InstanceOfName Inventer_Control
"Inventer_Control"
BEGIN
   ID := 6;
END_DATA_BLOCK

DATA_BLOCK "DETECT_VALUE"   // DB20
{ S7_Optimized_Access := 'FALSE' }
VERSION : 0.1
   VAR
      SCANED_BARCODE : String[10];
      INPUT_SCANED_BARCODE : String[10];
   END_VAR
BEGIN
END_DATA_BLOCK

DATA_BLOCK "Tranfer_2"   // DB21
{ S7_Optimized_Access := 'TRUE' }
VERSION : 0.1
// stored: InstanceOfName Inventer_Control
"Inventer_Control"
BEGIN
   ID := 7;
END_DATA_BLOCK

DATA_BLOCK "DATA_TEMPERATER"   // DB24
{ S7_Optimized_Access := 'FALSE' }
VERSION : 0.1
   VAR
      Nhiet_Do_Tank1 : Real;
      Nhiet_Do_Tank2 : Real;
      Nhiet_Do_Tank3 : Real;
      Nhiet_Do_Tank4 : Real;
      Nhiet_Do_Tank5 : Real;
      Nhiet_Do_Tank6 : Real;
      Nhiet_Do_Tank7 : Real;
      Nhiet_Do_Tank8 : Real;
      Nhiet_Do_Tank9 : Real;
      Nhiet_Do_Tank10 : Real;
      Nhiet_Do_Tank11 : Real;
   END_VAR
BEGIN
END_DATA_BLOCK

DATA_BLOCK "MB_Comunicate"   // DB136
{ S7_Optimized_Access := 'FALSE' }
VERSION : 0.1
   VAR
      Req : Bool;
      Error : Bool;
      Done : Bool;
      Busy : Bool;
      Status : Word;
      DataPtr : Array[0..8] of Int;
      DataLen : Int;
      MB_ID : UInt;
      Mode : UInt;
      DataAddr : UDInt;
      Device : Int;
   END_VAR
BEGIN
END_DATA_BLOCK

// folder: System blocks/Program resources

DATA_BLOCK "PLC_1_Connection_DB"   // DB4
{ S7_Optimized_Access := 'TRUE' }
AUTHOR : SIMATIC
FAMILY : MC7Plus
NAME : TC_IP_v4
VERSION : 1.0
// stored: InstanceOfName TCON_IP_v4
"TCON_IP_v4"
BEGIN
   ID := 1;
   InterfaceId := 64;
   LocalPort := 2000;
   RemotePort := 2000;
   ActiveEstablished := true;
   RemoteAddress.ADDR[1] := 192;
   RemoteAddress.ADDR[2] := 168;
   RemoteAddress.ADDR[4] := 3;
END_DATA_BLOCK

DATA_BLOCK "Reset_delay"   // DB22
{ S7_Optimized_Access := 'TRUE' }
AUTHOR : Simatic
FAMILY : IEC
NAME : IEC_TMR
VERSION : 1.0
// stored: InstanceOfName IEC_TIMER
"IEC_TIMER"
BEGIN
END_DATA_BLOCK

DATA_BLOCK "delay_return_home _1"   // DB23
{ S7_Optimized_Access := 'TRUE' }
AUTHOR : Simatic
FAMILY : IEC
NAME : IEC_TMR
VERSION : 1.0
// stored: InstanceOfName IEC_TIMER
"IEC_TIMER"
BEGIN
END_DATA_BLOCK

DATA_BLOCK "Delay_1s"   // DB25
{ S7_Optimized_Access := 'TRUE' }
AUTHOR : Simatic
FAMILY : IEC
NAME : IEC_TMR
VERSION : 1.0
// stored: InstanceOfName IEC_TIMER
"IEC_TIMER"
BEGIN
END_DATA_BLOCK

DATA_BLOCK "Delay_1s_1"   // DB26
{ S7_Optimized_Access := 'TRUE' }
AUTHOR : Simatic
FAMILY : IEC
NAME : IEC_TMR
VERSION : 1.0
// stored: InstanceOfName IEC_TIMER
"IEC_TIMER"
BEGIN
END_DATA_BLOCK

DATA_BLOCK "Delay_1s_2"   // DB27
{ S7_Optimized_Access := 'TRUE' }
AUTHOR : Simatic
FAMILY : IEC
NAME : IEC_TMR
VERSION : 1.0
// stored: InstanceOfName IEC_TIMER
"IEC_TIMER"
BEGIN
END_DATA_BLOCK

DATA_BLOCK "Time_Tripping_Area1"   // DB28
{ S7_Optimized_Access := 'TRUE' }
AUTHOR : Simatic
FAMILY : IEC
NAME : IEC_TMR
VERSION : 1.0
// stored: InstanceOfName IEC_TIMER
"IEC_TIMER"
BEGIN
END_DATA_BLOCK

DATA_BLOCK "Delay_1s_3"   // DB29
{ S7_Optimized_Access := 'TRUE' }
AUTHOR : Simatic
FAMILY : IEC
NAME : IEC_TMR
VERSION : 1.0
// stored: InstanceOfName IEC_TIMER
"IEC_TIMER"
BEGIN
END_DATA_BLOCK

DATA_BLOCK "Delay_1s_4"   // DB30
{ S7_Optimized_Access := 'TRUE' }
AUTHOR : Simatic
FAMILY : IEC
NAME : IEC_TMR
VERSION : 1.0
// stored: InstanceOfName IEC_TIMER
"IEC_TIMER"
BEGIN
END_DATA_BLOCK

DATA_BLOCK "Delay_1s_5"   // DB31
{ S7_Optimized_Access := 'TRUE' }
AUTHOR : Simatic
FAMILY : IEC
NAME : IEC_TMR
VERSION : 1.0
// stored: InstanceOfName IEC_TIMER
"IEC_TIMER"
BEGIN
END_DATA_BLOCK

DATA_BLOCK "Delay_1s_6"   // DB32
{ S7_Optimized_Access := 'TRUE' }
AUTHOR : Simatic
FAMILY : IEC
NAME : IEC_TMR
VERSION : 1.0
// stored: InstanceOfName IEC_TIMER
"IEC_TIMER"
BEGIN
END_DATA_BLOCK

DATA_BLOCK "Delay_1s_7"   // DB33
{ S7_Optimized_Access := 'TRUE' }
AUTHOR : Simatic
FAMILY : IEC
NAME : IEC_TMR
VERSION : 1.0
// stored: InstanceOfName IEC_TIMER
"IEC_TIMER"
BEGIN
END_DATA_BLOCK

DATA_BLOCK "delay_return_home _2"   // DB34
{ S7_Optimized_Access := 'TRUE' }
AUTHOR : Simatic
FAMILY : IEC
NAME : IEC_TMR
VERSION : 1.0
// stored: InstanceOfName IEC_TIMER
"IEC_TIMER"
BEGIN
END_DATA_BLOCK

DATA_BLOCK "delay_return_home _3"   // DB35
{ S7_Optimized_Access := 'TRUE' }
AUTHOR : Simatic
FAMILY : IEC
NAME : IEC_TMR
VERSION : 1.0
// stored: InstanceOfName IEC_TIMER
"IEC_TIMER"
BEGIN
END_DATA_BLOCK

DATA_BLOCK "delay_return_home _4"   // DB36
{ S7_Optimized_Access := 'TRUE' }
AUTHOR : Simatic
FAMILY : IEC
NAME : IEC_TMR
VERSION : 1.0
// stored: InstanceOfName IEC_TIMER
"IEC_TIMER"
BEGIN
END_DATA_BLOCK

DATA_BLOCK "Delay_4s"   // DB37
{ S7_Optimized_Access := 'TRUE' }
AUTHOR : Simatic
FAMILY : IEC
NAME : IEC_TMR
VERSION : 1.0
// stored: InstanceOfName IEC_TIMER
"IEC_TIMER"
BEGIN
END_DATA_BLOCK

DATA_BLOCK "Delay_2_5s"   // DB38
{ S7_Optimized_Access := 'TRUE' }
AUTHOR : Simatic
FAMILY : IEC
NAME : IEC_TMR
VERSION : 1.0
// stored: InstanceOfName IEC_TIMER
"IEC_TIMER"
BEGIN
END_DATA_BLOCK

DATA_BLOCK "tee"   // DB39
{ S7_Optimized_Access := 'TRUE' }
AUTHOR : Simatic
FAMILY : IEC
NAME : CNTR
VERSION : 1.0
// stored: InstanceOfName IEC_COUNTER
"IEC_COUNTER"
BEGIN
END_DATA_BLOCK

DATA_BLOCK "After_Done_Trip_1"   // DB41
{ S7_Optimized_Access := 'TRUE' }
AUTHOR : Simatic
FAMILY : IEC
NAME : IEC_TMR
VERSION : 1.0
// stored: InstanceOfName IEC_TIMER
"IEC_TIMER"
BEGIN
END_DATA_BLOCK

DATA_BLOCK "After_Done_Trip_3"   // DB42
{ S7_Optimized_Access := 'TRUE' }
AUTHOR : Simatic
FAMILY : IEC
NAME : IEC_TMR
VERSION : 1.0
// stored: InstanceOfName IEC_TIMER
"IEC_TIMER"
BEGIN
END_DATA_BLOCK

DATA_BLOCK "Delay_Down_Robot"   // DB43
{ S7_Optimized_Access := 'TRUE' }
AUTHOR : Simatic
FAMILY : IEC
NAME : IEC_TMR
VERSION : 1.0
// stored: InstanceOfName IEC_TIMER
"IEC_TIMER"
BEGIN
END_DATA_BLOCK

DATA_BLOCK "Delay_Kẹp"   // DB44
{ S7_Optimized_Access := 'TRUE' }
AUTHOR : Simatic
FAMILY : IEC
NAME : IEC_TMR
VERSION : 1.0
// stored: InstanceOfName IEC_TIMER
"IEC_TIMER"
BEGIN
END_DATA_BLOCK

DATA_BLOCK "Delay_Up_XL_Robot"   // DB45
{ S7_Optimized_Access := 'TRUE' }
AUTHOR : Simatic
FAMILY : IEC
NAME : IEC_TMR
VERSION : 1.0
// stored: InstanceOfName IEC_TIMER
"IEC_TIMER"
BEGIN
END_DATA_BLOCK

DATA_BLOCK "Delay_Move_to_P2_Robot"   // DB46
{ S7_Optimized_Access := 'TRUE' }
AUTHOR : Simatic
FAMILY : IEC
NAME : IEC_TMR
VERSION : 1.0
// stored: InstanceOfName IEC_TIMER
"IEC_TIMER"
BEGIN
END_DATA_BLOCK

DATA_BLOCK "Delay_Down_Robot_P2"   // DB47
{ S7_Optimized_Access := 'TRUE' }
AUTHOR : Simatic
FAMILY : IEC
NAME : IEC_TMR
VERSION : 1.0
// stored: InstanceOfName IEC_TIMER
"IEC_TIMER"
BEGIN
END_DATA_BLOCK

DATA_BLOCK "Delay_Open_XL_Kẹp"   // DB48
{ S7_Optimized_Access := 'TRUE' }
AUTHOR : Simatic
FAMILY : IEC
NAME : IEC_TMR
VERSION : 1.0
// stored: InstanceOfName IEC_TIMER
"IEC_TIMER"
BEGIN
END_DATA_BLOCK

DATA_BLOCK "Delay_Up_XL_Robot_1"   // DB49
{ S7_Optimized_Access := 'TRUE' }
AUTHOR : Simatic
FAMILY : IEC
NAME : IEC_TMR
VERSION : 1.0
// stored: InstanceOfName IEC_TIMER
"IEC_TIMER"
BEGIN
END_DATA_BLOCK

DATA_BLOCK "Delay_Move_to_PStart_Robot"   // DB50
{ S7_Optimized_Access := 'TRUE' }
AUTHOR : Simatic
FAMILY : IEC
NAME : IEC_TMR
VERSION : 1.0
// stored: InstanceOfName IEC_TIMER
"IEC_TIMER"
BEGIN
END_DATA_BLOCK

DATA_BLOCK "Time_Tripping_Area3"   // DB51
{ S7_Optimized_Access := 'TRUE' }
AUTHOR : Simatic
FAMILY : IEC
NAME : IEC_TMR
VERSION : 1.0
// stored: InstanceOfName IEC_TIMER
"IEC_TIMER"
BEGIN
END_DATA_BLOCK

DATA_BLOCK "Timer_Trip_Area_Robot"   // DB52
{ S7_Optimized_Access := 'TRUE' }
AUTHOR : Simatic
FAMILY : IEC
NAME : IEC_TMR
VERSION : 1.0
// stored: InstanceOfName IEC_TIMER
"IEC_TIMER"
BEGIN
END_DATA_BLOCK

DATA_BLOCK "Delay_to_Active_Robot"   // DB53
{ S7_Optimized_Access := 'TRUE' }
AUTHOR : Simatic
FAMILY : IEC
NAME : IEC_TMR
VERSION : 1.0
// stored: InstanceOfName IEC_TIMER
"IEC_TIMER"
BEGIN
END_DATA_BLOCK

DATA_BLOCK "Timer_Run_FW_Conveyor_Input"   // DB54
{ S7_Optimized_Access := 'TRUE' }
AUTHOR : Simatic
FAMILY : IEC
NAME : IEC_TMR
VERSION : 1.0
// stored: InstanceOfName IEC_TIMER
"IEC_TIMER"
BEGIN
END_DATA_BLOCK

DATA_BLOCK "Timer_run_BW_Conveyor_Input"   // DB55
{ S7_Optimized_Access := 'TRUE' }
AUTHOR : Simatic
FAMILY : IEC
NAME : IEC_TMR
VERSION : 1.0
// stored: InstanceOfName IEC_TIMER
"IEC_TIMER"
BEGIN
END_DATA_BLOCK

DATA_BLOCK "Delay_1s_8"   // DB56
{ S7_Optimized_Access := 'TRUE' }
AUTHOR : Simatic
FAMILY : IEC
NAME : IEC_TMR
VERSION : 1.0
// stored: InstanceOfName IEC_TIMER
"IEC_TIMER"
BEGIN
END_DATA_BLOCK

DATA_BLOCK "Timer_Delay_Up_LIFT_2"   // DB57
{ S7_Optimized_Access := 'TRUE' }
AUTHOR : Simatic
FAMILY : IEC
NAME : IEC_TMR
VERSION : 1.0
// stored: InstanceOfName IEC_TIMER
"IEC_TIMER"
BEGIN
END_DATA_BLOCK

DATA_BLOCK "wait_reset_1"   // DB134
{ S7_Optimized_Access := 'TRUE' }
AUTHOR : Simatic
FAMILY : IEC
NAME : IEC_TMR
VERSION : 1.0
// stored: InstanceOfName IEC_TIMER
"IEC_TIMER"
BEGIN
END_DATA_BLOCK

DATA_BLOCK "Check_timeout"   // DB135
{ S7_Optimized_Access := 'TRUE' }
AUTHOR : Simatic
FAMILY : IEC
NAME : IEC_TMR
VERSION : 1.0
// stored: InstanceOfName IEC_TIMER
"IEC_TIMER"
BEGIN
END_DATA_BLOCK

// folder: (top level)

FUNCTION_BLOCK "MB_Axis"   // FB8, LAD
{ S7_Optimized_Access := 'TRUE' }
VERSION : 0.1
   VAR_INPUT
      Busy : Bool;
      Done : Bool;
      Error : Bool;
      Status : Word;
      Enable_block : Bool;
   END_VAR
   VAR_OUTPUT
      Req : Bool;
      Mb_ID : UInt;
      DataLen : UInt := 1;
      DataAddr : UDInt;
      Mode : UInt;
   END_VAR
   VAR_IN_OUT
      Ptr : Array[0..8] of Int;
   END_VAR
   VAR
      Process : "Process";
   END_VAR
   VAR RETAIN
      MasterData : "MasterData";
      Jog_Speed : Int := 200;
      Home_Speed : Int := 100;
   END_VAR
   VAR
      Select_Point : Int := 1;
      "Jog-" : Bool;
      "Jog+" : Bool;
      "Find Home" : Bool;
      Set_point : Bool;
      Enable_Ser : Bool;
      Disable_Ser : Bool;
      Move_point : Bool;
      "RW Done" : Bool;
      HOME : Bool;
      Enable_Write : Bool;
      "DisJog-" : Bool;
      "DisJog+" : Bool;
      Home_excuting : Bool;
      Reset_fault : Bool;
      "Enable Read" : Bool;
      Home_Done : Bool;
      Move_point_done : Bool;
      Move_Absolute : Bool;
      temp1 : Bool;
      temp2 : Bool;
      Reset_Servo : Bool;
      Set_home : Bool;
      All_Done : Bool := true;
      Sensor_home : Bool;
      Write_Full_Done : Bool := true;
      Read_Full_Done : Bool := true;
      Wait_lost_sensor : Bool;
      Re_home_Excuting : Bool;
      Wait_lost_sensor_1 : Bool;
      Check_reHome : Bool;
      Re_home : Bool;
      Mode_Home : Bool;
      Trigger_home_done : Bool;
      Out_Range_Home : Bool;
      delay_rs : Time := T#400ms;
      Trigger_home_done_1 : Bool;
      temp3 : Bool;
      Sensor_Limit : Bool;
      Delay_Home_Done : Bool;
      Jog_FW_Home_Excuting : Bool;
      Move_Home : Bool;
      Finding : Bool;
      Home_begin : Bool;
      EMG_STOP : Bool;
   END_VAR
   VAR_TEMP   // added for the SCL form of the ladder/FBD networks
      _w1 : Bool;
      _w2 : Bool;
      _w3 : Bool;
      _w4 : Bool;
      _w5 : Bool;
      _w6 : Bool;
      _w7 : Bool;
      _w8 : Bool;
      _w9 : Bool;
      _w10 : Bool;
      _w11 : Bool;
      _w12 : Bool;
      _w13 : Bool;
      _w14 : Bool;
      _w15 : Bool;
   END_VAR
BEGIN

REGION Network 1 (SCL)
   IF #Process.Step = 1 THEN
       ;
       #Process.mobusMaster.Mode := 2;
       #Mode := #Process.mobusMaster.Mode;
       #Process.mobusMaster.MbAddress := #MasterData.ID;
       #Mb_ID := INT_TO_UINT(#Process.mobusMaster.MbAddress);
       IF #Process.Step_W = 1 THEN
           ;
           #Process.mobusMaster.DataAddr := 424641;
           #DataAddr := #Process.mobusMaster.DataAddr;
       ELSIF #Process.Step_W = 2 THEN
           ;
           #Process.mobusMaster.DataAddr := 424673;
           #DataAddr := #Process.mobusMaster.DataAddr;
       ELSIF #Process.Step_W = 3 THEN
           ;
           #Process.mobusMaster.DataAddr := 424706;
           #DataAddr := #Process.mobusMaster.DataAddr;
       ELSIF #Process.Step_W = 4 THEN
           ;
           #Process.mobusMaster.DataAddr := 411617;
           #DataAddr := #Process.mobusMaster.DataAddr;
       ELSIF #Process.Step_W = 5 THEN
           ;
           #Process.mobusMaster.DataAddr := 424641;
           #DataAddr := #Process.mobusMaster.DataAddr;
       ELSIF #Process.Step_W = 6 THEN
           ;
           #Process.mobusMaster.DataAddr := 424729;
           #DataAddr := #Process.mobusMaster.DataAddr;
       ELSIF #Process.Step_W = 11 THEN
           ;
           #Process.mobusMaster.DataAddr := 410242;
           #DataAddr := #Process.mobusMaster.DataAddr;
       ELSIF #Process.Step_W = 12 THEN
           ;
           #Process.mobusMaster.DataAddr := 410243;
           #DataAddr := #Process.mobusMaster.DataAddr;
       ELSIF #Process.Step_W = 13 THEN
           ;
           #Process.mobusMaster.DataAddr := 410244;
           #DataAddr := #Process.mobusMaster.DataAddr;
       ELSIF #Process.Step_W = 14 THEN
           ;
           #Process.mobusMaster.DataAddr := 410245;
           #DataAddr := #Process.mobusMaster.DataAddr;
       ELSIF #Process.Step_W = 15 THEN
           ;
           #Process.mobusMaster.DataAddr := 410246;
           #DataAddr := #Process.mobusMaster.DataAddr;
       ELSIF #Process.Step_W = 16 THEN
           ;
           #Process.mobusMaster.DataAddr := 410247;
           #DataAddr := #Process.mobusMaster.DataAddr;
       ELSIF #Process.Step_W = 17 THEN
           ;
           #Process.mobusMaster.DataAddr := 410248;
           #DataAddr := #Process.mobusMaster.DataAddr;
       ELSIF #Process.Step_W = 18 THEN
           ;
           #Process.mobusMaster.DataAddr := 410249;
           #DataAddr := #Process.mobusMaster.DataAddr;
       ELSIF #Process.Step_W = 19 THEN
           ;
           #Process.mobusMaster.DataAddr := 410250;
           #DataAddr := #Process.mobusMaster.DataAddr;
       ELSIF #Process.Step_W = 20 THEN
           ;
           #Process.mobusMaster.DataAddr := 410251;
           #DataAddr := #Process.mobusMaster.DataAddr;
       ELSIF #Process.Step_W = 21 THEN
           ;
           #Process.mobusMaster.DataAddr := 410252;
           #DataAddr := #Process.mobusMaster.DataAddr;
       ELSIF #Process.Step_W = 22 THEN
           ;
           #Process.mobusMaster.DataAddr := 410253;
           #DataAddr := #Process.mobusMaster.DataAddr;
       ELSIF #Process.Step_W = 23 THEN
           ;
           #Process.mobusMaster.DataAddr := 410254;
           #DataAddr := #Process.mobusMaster.DataAddr;
       ELSIF #Process.Step_W = 24 THEN
           ;
           #Process.mobusMaster.DataAddr := 410255;
           #DataAddr := #Process.mobusMaster.DataAddr;
       ELSIF #Process.Step_W = 25 THEN
           ;
           #Process.mobusMaster.DataAddr := 410256;
           #DataAddr := #Process.mobusMaster.DataAddr;
       ELSIF #Process.Step_W = 26 THEN
           ;
           #Process.mobusMaster.DataAddr := 410257;
           #DataAddr := #Process.mobusMaster.DataAddr;
       ELSIF #Process.Step_W = 27 THEN
           ;
           #Process.mobusMaster.DataAddr := 410258;
           #DataAddr := #Process.mobusMaster.DataAddr;
       ELSIF #Process.Step_W = 28 THEN
           ;
           #Process.mobusMaster.DataAddr := 410259;
           #DataAddr := #Process.mobusMaster.DataAddr;
       ELSIF #Process.Step_W = 29 THEN
           ;
           #Process.mobusMaster.DataAddr := 410260;
           #DataAddr := #Process.mobusMaster.DataAddr;
       ELSIF #Process.Step_W = 30 THEN
           ;
           #Process.mobusMaster.DataAddr := 410261;
           #DataAddr := #Process.mobusMaster.DataAddr;
       ELSIF #Process.Step_W = 31 THEN
           ;
           #Process.mobusMaster.DataAddr := 410262;
           #DataAddr := #Process.mobusMaster.DataAddr;
       ELSIF #Process.Step_W = 32 THEN
           ;
           #Process.mobusMaster.DataAddr := 410263;
           #DataAddr := #Process.mobusMaster.DataAddr;
       ELSIF #Process.Step_W = 33 THEN
           ;
           #Process.mobusMaster.DataAddr := 410264;
           #DataAddr := #Process.mobusMaster.DataAddr;
       ELSIF #Process.Step_W = 34 THEN
           ;
           #Process.mobusMaster.DataAddr := 410265;
           #DataAddr := #Process.mobusMaster.DataAddr;
       ELSIF #Process.Step_W = 35 THEN
           ;
           #Process.mobusMaster.DataAddr := 410266;
           #DataAddr := #Process.mobusMaster.DataAddr;
       ELSIF #Process.Step_W = 36 THEN
           ;
           #Process.mobusMaster.DataAddr := 410267;
           #DataAddr := #Process.mobusMaster.DataAddr;
       ELSIF #Process.Step_W = 37 THEN
           ;
           #Process.mobusMaster.DataAddr := 410268;
           #DataAddr := #Process.mobusMaster.DataAddr;
       ELSIF #Process.Step_W = 38 THEN
           ;
           #Process.mobusMaster.DataAddr := 410269;
           #DataAddr := #Process.mobusMaster.DataAddr;
       ELSIF #Process.Step_W = 39 THEN
           ;
           #Process.mobusMaster.DataAddr := 410270;
           #DataAddr := #Process.mobusMaster.DataAddr;
       ELSIF #Process.Step_W = 40 THEN
           ;
           #Process.mobusMaster.DataAddr := 410271;
           #DataAddr := #Process.mobusMaster.DataAddr;
       END_IF;

       #MasterData.SendData := #Process.SinggleData;
       IF #Process.Step_W <10 & #Process.Step_W <> 3 THEN
           ;
           #Process.mobusMaster.DataLen := 1;
           #DataLen := #Process.mobusMaster.DataLen;
       ELSIF #Process.Step_W < 10 & #Process.Step_W = 3 THEN
           ;
           #Process.mobusMaster.DataLen := 2;
           #DataLen := #Process.mobusMaster.DataLen;
       ELSE
           ;
           #Process.mobusMaster.DataLen := 6;
           #DataLen := #Process.mobusMaster.DataLen;
       END_IF;

       #MasterData.DataPtr := #MasterData.SendData;
       #Ptr := #MasterData.DataPtr;

       #Process.mobusMaster.Req := TRUE;

       IF #Process.mobusMaster.Busy THEN
           ;
           #Process.Step := 2;
       END_IF;

   ELSIF #Process.Step = 2 THEN
       ;
       IF #Process.mobusMaster.Done THEN
           ;
           #Process.mobusMaster.Req := FALSE;
           #Process.Step := 5;
       END_IF;
   ELSIF #Process.Step = 3 THEN
       ;
       #Process.mobusMaster.Mode := 0;
       #Mode := #Process.mobusMaster.Mode;
       #Process.mobusMaster.MbAddress := #MasterData.ID;
       #Mb_ID := INT_TO_UINT(#Process.mobusMaster.MbAddress);
       IF #Process.Step_R = 1 THEN
           ;
           #Process.mobusMaster.DataAddr := 424642;
           #DataAddr := #Process.mobusMaster.DataAddr;
           #Process.mobusMaster.DataLen := 1;
           #DataLen := #Process.mobusMaster.DataLen;
       ELSIF #Process.Step_R = 2 THEN
           ;
           #Process.mobusMaster.DataAddr := 411056;
           #DataAddr := #Process.mobusMaster.DataAddr;
           #Process.mobusMaster.DataLen := 2;
           #DataLen := #Process.mobusMaster.DataLen;
       ELSIF #Process.Step_R = 3 THEN
           ;
           #Process.mobusMaster.DataAddr := 411625;
           #DataAddr := #Process.mobusMaster.DataAddr;
           #Process.mobusMaster.DataLen := 2;
           #DataLen := #Process.mobusMaster.DataLen;
       ELSIF #Process.Step_R = 4 THEN
           ;
           #Process.mobusMaster.DataAddr := 424706;
           #DataAddr := #Process.mobusMaster.DataAddr;
           #Process.mobusMaster.DataLen := 2;
           #DataLen := #Process.mobusMaster.DataLen;
       END_IF;

       #Process.mobusMaster.Req := TRUE;
       IF #Process.mobusMaster.Busy = TRUE THEN
           ;
           #Process.Step := 4;
       END_IF;
   ELSIF #Process.Step = 4 & #Process.mobusMaster.Done = TRUE THEN
       ;
       #Process.mobusMaster.Req := FALSE;

       IF #Process.Step_R = 1  THEN
           ;
           #MasterData.ReceivedData := #Ptr;
           #MasterData.Status := #MasterData.ReceivedData[0];
           "INT_TO_BIT_ARRAY"(IN := #MasterData.Status,
                              OUT => #MasterData.Array_Status);
       ELSIF #Process.Step_R = 2 THEN
           ;
           #MasterData.ReceivedData := #Ptr;
           #MasterData.Current_Position[0] := #MasterData.ReceivedData[0];
           #MasterData.Current_Position[1] := #MasterData.ReceivedData[1];

       ELSIF #Process.Step_R = 3 THEN
           ;
           #MasterData.ReceivedData := #Ptr;
           #MasterData.Current_Table_Point[0] := #MasterData.ReceivedData[0];
           #MasterData.Current_Table_Point[1] := #MasterData.ReceivedData[1];
       ELSIF #Process.Step_R = 4 THEN
           ;
           #MasterData.ReceivedData := #Ptr;
           #MasterData.Current_Speed[0] := #MasterData.ReceivedData[0];
           #MasterData.Current_Speed[1] := #MasterData.ReceivedData[1];
       END_IF;
       #Process.Step := 5;
       END_IF;
END_REGION

REGION Network 2: Input pin
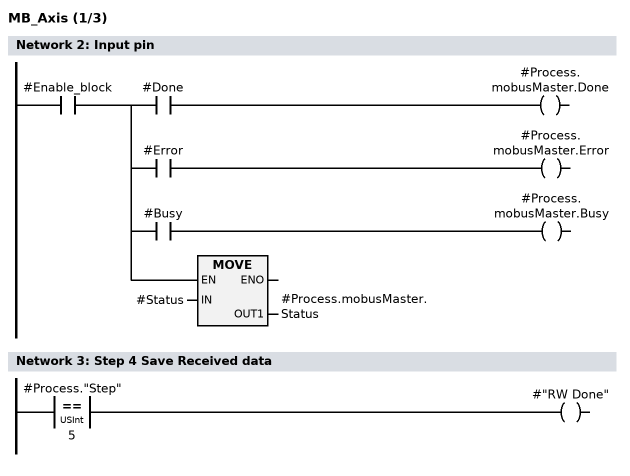
   RUNG wire#powerrail
      Contact( #Enable_block )
      wire#w1
      Contact( #Done )
      Coil( #Process.mobusMaster.Done )
   END_RUNG
   RUNG wire#w1
      Contact( #Error )
      Coil( #Process.mobusMaster.Error )
   END_RUNG
   RUNG wire#w1
      Contact( #Busy )
      Coil( #Process.mobusMaster.Busy )
   END_RUNG
   RUNG wire#w1
      Move(in := #Status, out1 => #Process.mobusMaster.Status)
   END_RUNG
   // the same network as SCL:
   #Process.mobusMaster.Done := #Enable_block AND #Done;
   #Process.mobusMaster.Error := #Enable_block AND #Error;
   #Process.mobusMaster.Busy := #Enable_block AND #Busy;
   IF #Enable_block THEN #Process.mobusMaster.Status := #Status; END_IF;
END_REGION

REGION Network 3: Step 4 Save Received data
   RUNG wire#powerrail
      { S7_Templates := "SrcType := USInt" } EQ_Contact(in1 := #Process."Step", in2 := 5)
      Coil( #"RW Done" )
   END_RUNG
   // the same network as SCL:
   #"RW Done" := #Process."Step" = 5;
END_REGION

REGION Network 4: Excute Command
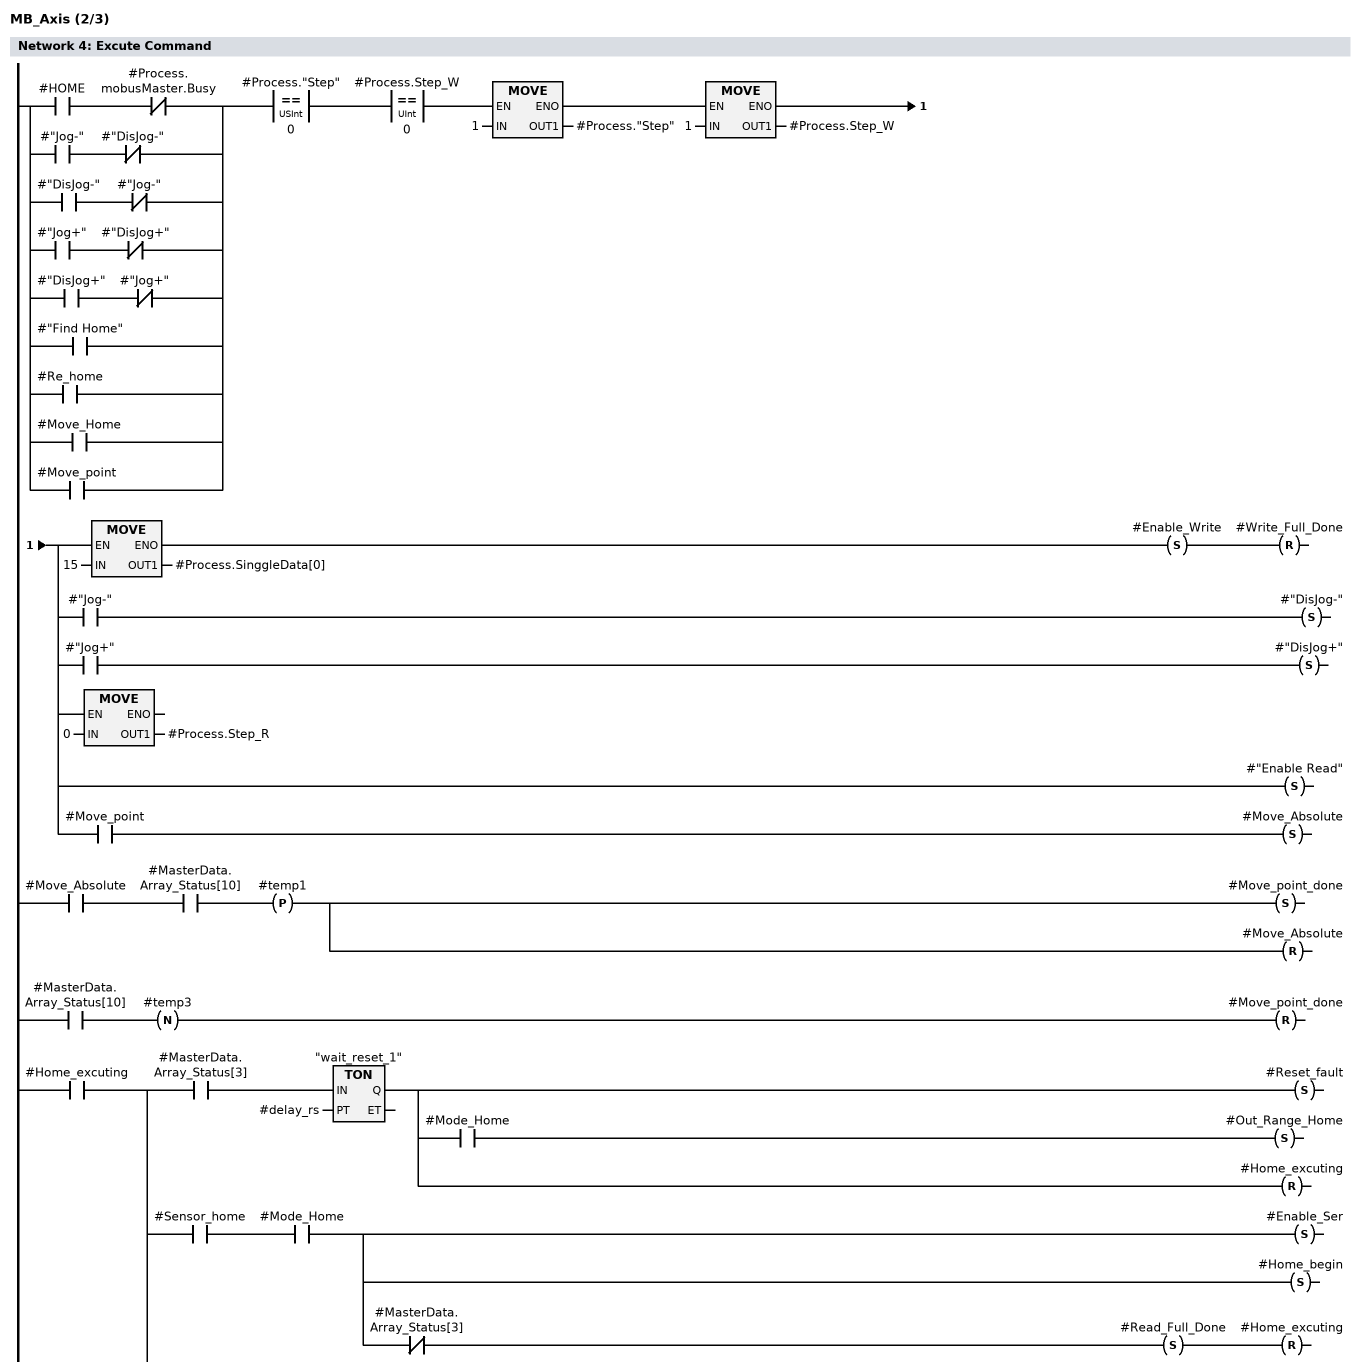
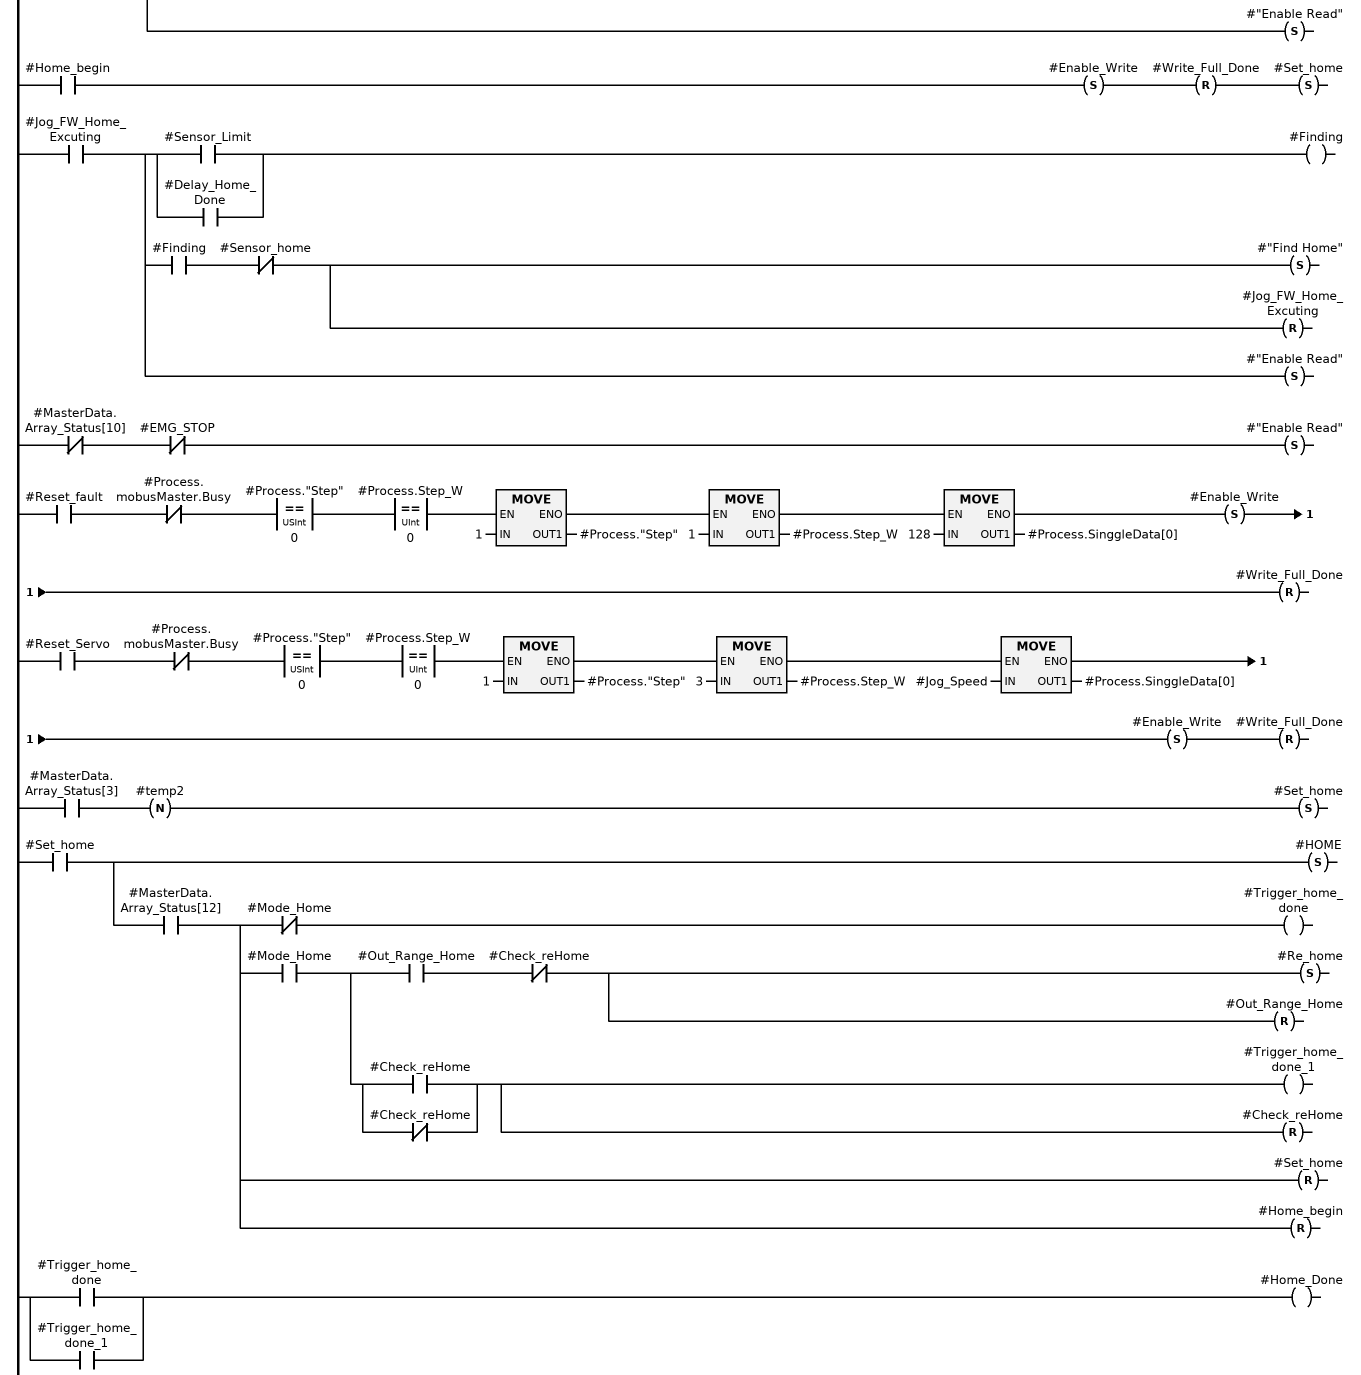
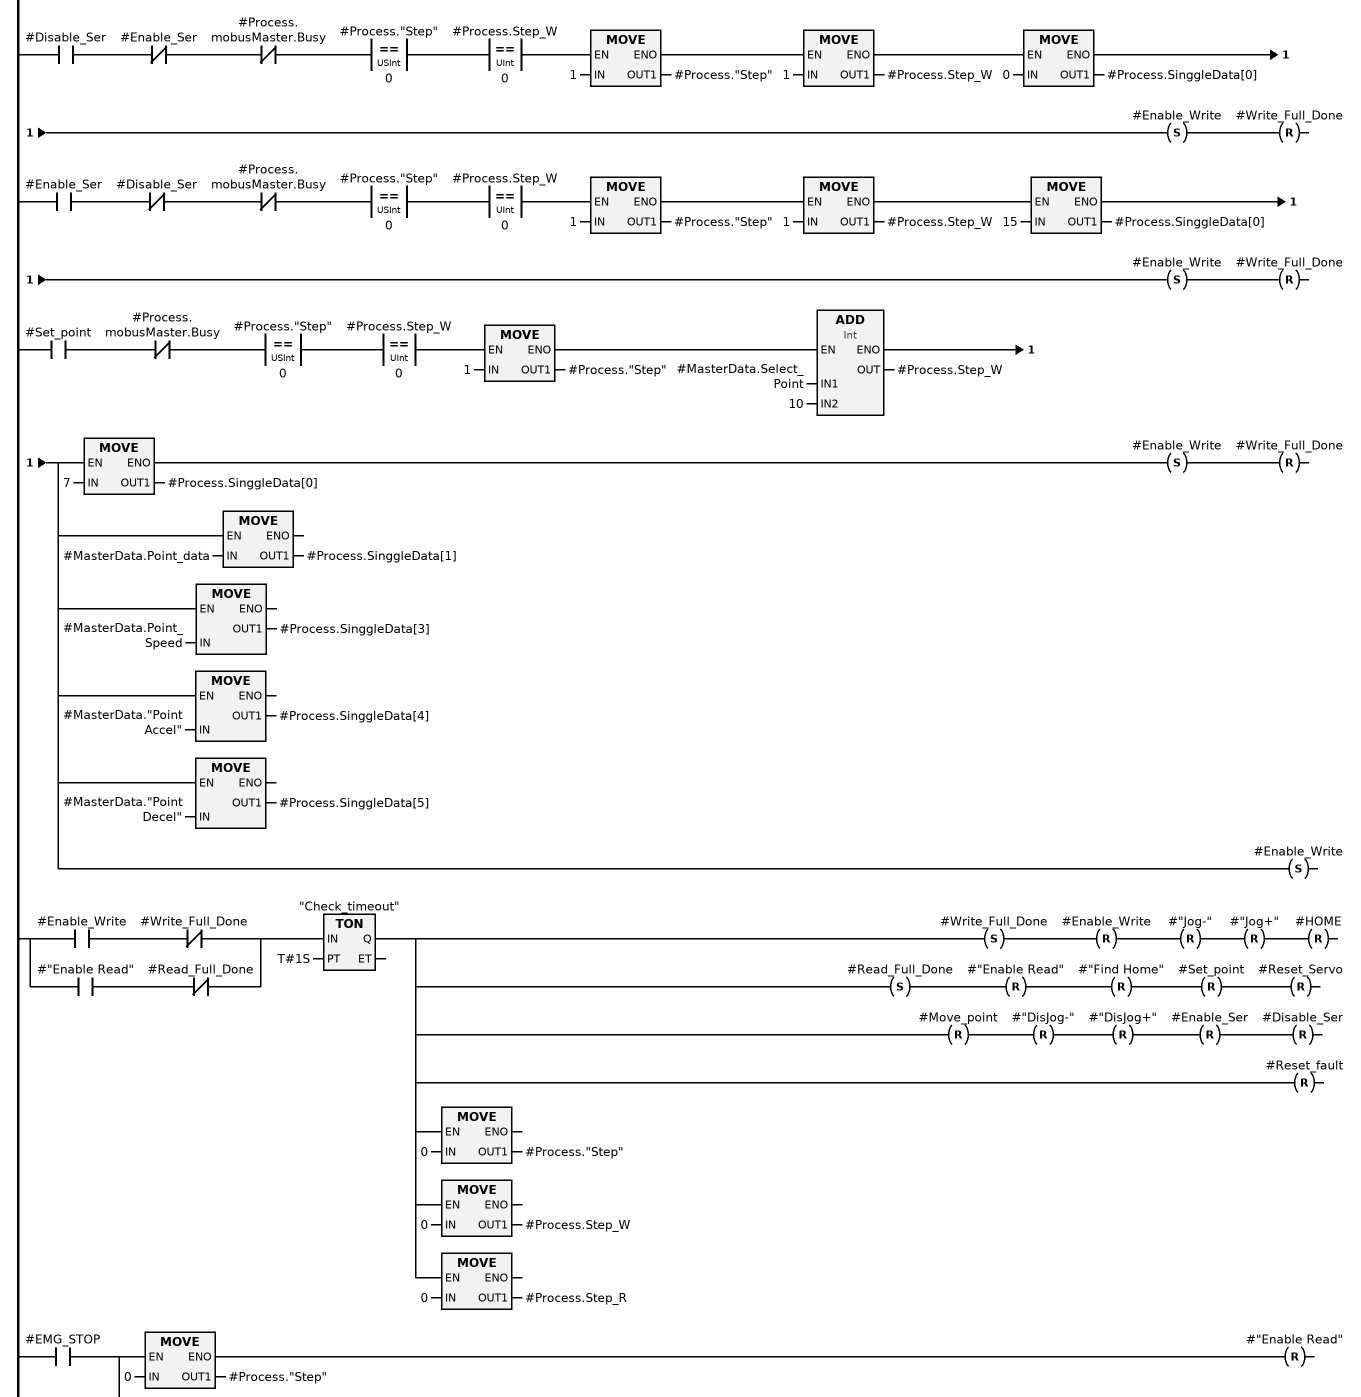
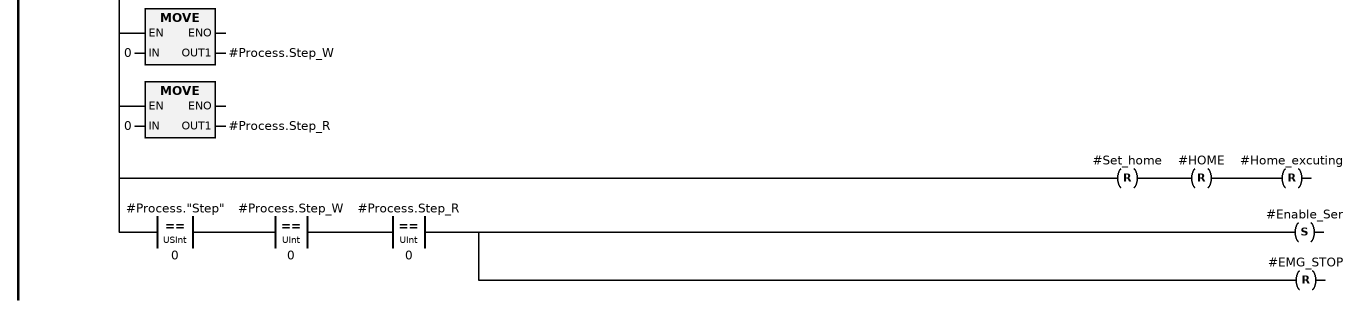
   #_w1 := ((#HOME AND NOT #Process.mobusMaster.Busy) OR (#"Jog-" AND NOT #"DisJog-") OR (#"DisJog-" AND NOT #"Jog-") OR (#"Jog+" AND NOT #"DisJog+") OR (#"DisJog+" AND NOT #"Jog+") OR #"Find Home" OR #Re_home OR #Move_Home OR #Move_point) AND (#Process."Step" = 0) AND (#Process.Step_W = 0);
   IF #_w1 THEN
       #Process."Step" := 1;
       #Process.Step_W := 1;
       #Process.SinggleData[0] := 15;
       #Enable_Write := TRUE;
       #Write_Full_Done := FALSE;
   END_IF;
   IF #_w1 AND #"Jog-" THEN #"DisJog-" := TRUE; END_IF;
   IF #_w1 AND #"Jog+" THEN #"DisJog+" := TRUE; END_IF;
   IF #_w1 THEN
       #Process.Step_R := 0;
       #"Enable Read" := TRUE;
   END_IF;
   IF #_w1 AND #Move_point THEN #Move_Absolute := TRUE; END_IF;
   #_w2 := #Move_Absolute AND #MasterData.Array_Status[10];
   #_w3 := #_w2 AND NOT #temp1;   // rising edge
   #temp1 := #_w2;
   IF #_w3 THEN
       #Move_point_done := TRUE;
       #Move_Absolute := FALSE;
   END_IF;
   #_w4 := NOT #MasterData.Array_Status[10] AND #temp3;   // falling edge
   #temp3 := #MasterData.Array_Status[10];
   IF #_w4 THEN #Move_point_done := FALSE; END_IF;
   "wait_reset_1".TON(IN := #Home_excuting AND #MasterData.Array_Status[3], PT := #delay_rs);
   IF "wait_reset_1".Q THEN #Reset_fault := TRUE; END_IF;
   IF "wait_reset_1".Q AND #Mode_Home THEN #Out_Range_Home := TRUE; END_IF;
   #_w5 := #Home_excuting;
   IF "wait_reset_1".Q THEN #Home_excuting := FALSE; END_IF;
   #_w6 := #_w5 AND #Sensor_home AND #Mode_Home;
   IF #_w6 THEN
       #Enable_Ser := TRUE;
       #Home_begin := TRUE;
   END_IF;
   IF #_w6 AND NOT #MasterData.Array_Status[3] THEN
       #Read_Full_Done := TRUE;
       #Home_excuting := FALSE;
   END_IF;
   IF #_w5 THEN #"Enable Read" := TRUE; END_IF;
   IF #Home_begin THEN
       #Enable_Write := TRUE;
       #Write_Full_Done := FALSE;
       #Set_home := TRUE;
   END_IF;
   #Finding := #Jog_FW_Home_Excuting AND (#Sensor_Limit OR #Delay_Home_Done);
   IF #Jog_FW_Home_Excuting AND #Finding AND NOT #Sensor_home THEN #"Find Home" := TRUE; END_IF;
   #_w7 := #Jog_FW_Home_Excuting;
   IF #Jog_FW_Home_Excuting AND #Finding AND NOT #Sensor_home THEN #Jog_FW_Home_Excuting := FALSE; END_IF;
   IF #_w7 THEN #"Enable Read" := TRUE; END_IF;
   IF NOT #MasterData.Array_Status[10] AND NOT #EMG_STOP THEN #"Enable Read" := TRUE; END_IF;
   #_w8 := #Reset_fault AND NOT #Process.mobusMaster.Busy AND (#Process."Step" = 0) AND (#Process.Step_W = 0);
   IF #_w8 THEN
       #Process."Step" := 1;
       #Process.Step_W := 1;
       #Process.SinggleData[0] := 128;
       #Enable_Write := TRUE;
       #Write_Full_Done := FALSE;
   END_IF;
   #_w9 := #Reset_Servo AND NOT #Process.mobusMaster.Busy AND (#Process."Step" = 0) AND (#Process.Step_W = 0);
   IF #_w9 THEN
       #Process."Step" := 1;
       #Process.Step_W := 3;
       #Process.SinggleData[0] := #Jog_Speed;
       #Enable_Write := TRUE;
       #Write_Full_Done := FALSE;
   END_IF;
   #_w10 := NOT #MasterData.Array_Status[3] AND #temp2;   // falling edge
   #temp2 := #MasterData.Array_Status[3];
   IF #_w10 THEN #Set_home := TRUE; END_IF;
   IF #Set_home THEN #HOME := TRUE; END_IF;
   #_w11 := #Set_home AND #MasterData.Array_Status[12];
   #Trigger_home_done := #_w11 AND NOT #Mode_Home;
   #_w12 := #_w11 AND #Mode_Home;
   IF #_w12 AND #Out_Range_Home AND NOT #Check_reHome THEN
       #Re_home := TRUE;
       #Out_Range_Home := FALSE;
   END_IF;
   #Trigger_home_done_1 := #_w12 AND (#Check_reHome OR NOT #Check_reHome);
   IF #Trigger_home_done_1 THEN #Check_reHome := FALSE; END_IF;
   IF #_w11 THEN
       #Set_home := FALSE;
       #Home_begin := FALSE;
   END_IF;
   #Home_Done := #Trigger_home_done OR #Trigger_home_done_1;
   #_w13 := #Disable_Ser AND NOT #Enable_Ser AND NOT #Process.mobusMaster.Busy AND (#Process."Step" = 0) AND (#Process.Step_W = 0);
   IF #_w13 THEN
       #Process."Step" := 1;
       #Process.Step_W := 1;
       #Process.SinggleData[0] := 0;
       #Enable_Write := TRUE;
       #Write_Full_Done := FALSE;
   END_IF;
   #_w14 := #Enable_Ser AND NOT #Disable_Ser AND NOT #Process.mobusMaster.Busy AND (#Process."Step" = 0) AND (#Process.Step_W = 0);
   IF #_w14 THEN
       #Process."Step" := 1;
       #Process.Step_W := 1;
       #Process.SinggleData[0] := 15;
       #Enable_Write := TRUE;
       #Write_Full_Done := FALSE;
   END_IF;
   #_w15 := #Set_point AND NOT #Process.mobusMaster.Busy AND (#Process."Step" = 0) AND (#Process.Step_W = 0);
   IF #_w15 THEN
       #Process."Step" := 1;
       #Process.Step_W := #MasterData.Select_Point + 10;
       #Process.SinggleData[0] := 7;
       #Enable_Write := TRUE;
       #Write_Full_Done := FALSE;
       #Process.SinggleData[1] := #MasterData.Point_data;
       #Process.SinggleData[3] := #MasterData.Point_Speed;
       #Process.SinggleData[4] := #MasterData."Point Accel";
       #Process.SinggleData[5] := #MasterData."Point Decel";
       #Enable_Write := TRUE;
   END_IF;
   "Check_timeout".TON(IN := (#Enable_Write AND NOT #Write_Full_Done) OR (#"Enable Read" AND NOT #Read_Full_Done),
                       PT := T#1S);
   IF "Check_timeout".Q THEN
       #Write_Full_Done := TRUE;
       #Enable_Write := FALSE;
       #"Jog-" := FALSE;
       #"Jog+" := FALSE;
       #HOME := FALSE;
       #Read_Full_Done := TRUE;
       #"Enable Read" := FALSE;
       #"Find Home" := FALSE;
       #Set_point := FALSE;
       #Reset_Servo := FALSE;
       #Move_point := FALSE;
       #"DisJog-" := FALSE;
       #"DisJog+" := FALSE;
       #Enable_Ser := FALSE;
       #Disable_Ser := FALSE;
       #Reset_fault := FALSE;
       #Process."Step" := 0;
       #Process.Step_W := 0;
       #Process.Step_R := 0;
   END_IF;
   IF #EMG_STOP THEN
       #Process."Step" := 0;
       #"Enable Read" := FALSE;
       #Process.Step_W := 0;
       #Process.Step_R := 0;
       #Set_home := FALSE;
       #HOME := FALSE;
       #Home_excuting := FALSE;
   END_IF;
   IF #EMG_STOP AND (#Process."Step" = 0) AND (#Process.Step_W = 0) AND (#Process.Step_R = 0) THEN
       #Enable_Ser := TRUE;
       #EMG_STOP := FALSE;
   END_IF;
END_REGION

REGION Network 5: Read Control
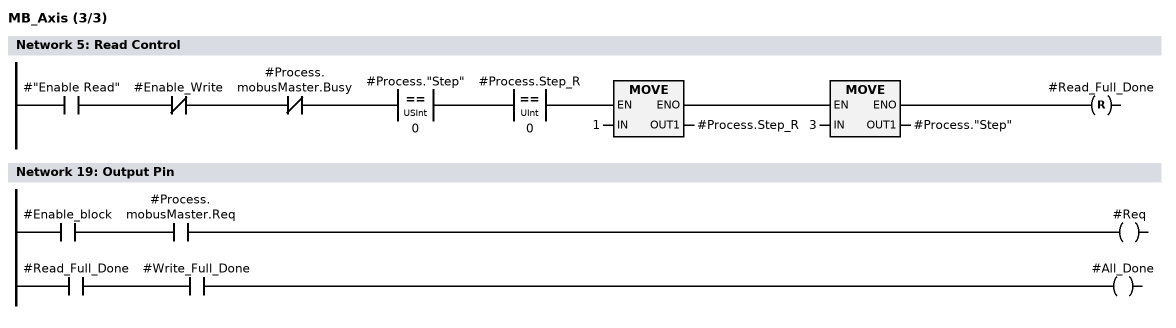
   RUNG wire#powerrail
      Contact( #"Enable Read" )
      I_Contact( #Enable_Write )
      I_Contact( #Process.mobusMaster.Busy )
      { S7_Templates := "SrcType := USInt" } EQ_Contact(in1 := #Process."Step", in2 := 0)
      { S7_Templates := "SrcType := UInt" } EQ_Contact(in1 := #Process.Step_R, in2 := 0)
      Move(in := 1, out1 => #Process.Step_R)
      Move(in := 3, out1 => #Process."Step")
      R_Coil( #Read_Full_Done )
   END_RUNG
   // the same network as SCL:
   #_w1 := #"Enable Read" AND NOT #Enable_Write AND NOT #Process.mobusMaster.Busy AND (#Process."Step" = 0) AND (#Process.Step_R = 0);
   IF #_w1 THEN
       #Process.Step_R := 1;
       #Process."Step" := 3;
       #Read_Full_Done := FALSE;
   END_IF;
END_REGION

REGION Network 6 (SCL): Read Process
   IF #"Enable Read"= TRUE & #"Process".mobusMaster.Busy = FALSE & #"RW Done"= TRUE & #"Enable_Write" = FALSE THEN
       ;
       IF #"Process".Step_R = 1 THEN
           #"Process".Step_R := 2;
           #"Process".Step := 3;
       ELSIF #"Process".Step_R = 2 THEN
           #"Process".Step_R := 3;
           #"Process".Step := 3;
       ELSIF #"Process".Step_R = 3 THEN
           #"Process".Step_R := 4;
           #"Process".Step := 3;
           // Done read Signed
       ELSIF #Process.Step_R = 4 THEN
           ;
           #Process.Step := 0;
           #Process.Step_R := 0;
           IF #MasterData.Array_Status[3] = TRUE & #Home_excuting = TRUE THEN
               ;
               #Read_Full_Done := FALSE;
           ELSE
               #Read_Full_Done := TRUE;
               ;
           END_IF;
           IF #MasterData.Array_Status[10] = TRUE THEN
               ;
               #"Enable Read" := FALSE;
           END_IF;
       END_IF;
   ELSIF #"Process".mobusMaster.Busy = FALSE &#"Process".Step_R <> 0 &#"RW Done" = TRUE &#"Enable_Write" = TRUE THEN
       ;
       #"Process".Step_R := 0;
       #"Process".Step := 0;
       #Read_Full_Done := TRUE;
   ELSIF #"Process".mobusMaster.Busy = FALSE &#"Process".Step_R <> 0 &#"Enable_Write" = FALSE &#"Enable Read" = FALSE &#"Process".Step <> 0 THEN
       ;
       #"Process".Step_R := 0;
       #"Process".Step := 0;
       #Read_Full_Done := TRUE;
   END_IF;
END_REGION

REGION Network 7 (SCL): Enable_Ser
   IF #"RW Done" = TRUE &#"Enable_Ser" = TRUE &#"Process".mobusMaster.Busy = FALSE THEN
       ;
       IF #"Process".Step_W = 1 THEN
           ;
           #"Process".Step_W := 0;
           #"Process".Step := 0;
           #"Enable_Ser" := FALSE;
           #"Enable Read" := TRUE;
           #Enable_Write := FALSE;
           #Write_Full_Done := TRUE;
           IF #Home_begin = TRUE THEN
               ;
               #Set_home := TRUE;
               #Home_begin := FALSE;

           END_IF;
           END_IF;
   END_IF;
END_REGION

REGION Network 8 (SCL): Disable_Ser
   IF #"RW Done" = TRUE &#"Disable_Ser" = TRUE &#"Process".mobusMaster.Busy = FALSE THEN
       ;
       IF #"Process".Step_W = 1 THEN
           ;
           #"Process".Step_W := 0;
           #"Process".Step := 0;
           #"Disable_Ser" := FALSE;
           #Enable_Write := FALSE;
           #Write_Full_Done := TRUE;
       END_IF;
   END_IF;
END_REGION

REGION Network 9 (SCL): Find Home
   IF #"RW Done" = TRUE &#"Find Home" = TRUE & #"Process".mobusMaster.Busy = FALSE THEN
       IF #"Process".Step_W = 1 THEN
           #"Process".Step_W := 2;
           #"Process".Step := 1;
           #"Process".SinggleData[0] := -100;
       ELSIF #"Process".Step_W = 2 THEN
           #"Process".Step_W := 3;
           #"Process".Step := 1;
           #"Process".SinggleData[0] := #Home_Speed;
           #Process.SinggleData[1] := 0;
       ELSIF #"Process".Step_W = 3 THEN
           #"Process".Step_W := 5;
           #"Process".Step := 1;
           #"Process".SinggleData[0] := 63;
           ;
       ELSIF #"Process".Step_W = 5 THEN
           #"Process".Step_W := 0;
           #"Process".Step := 0;
           #"Enable_Write" := FALSE;
           #"Home_excuting" := TRUE;
           #"Find Home" := FALSE;
           #Write_Full_Done := TRUE;
           // <Enable read to read Alarm>
           // 
           // Statement
           // 
           //<End>
           ;
       END_IF;
       ;
   END_IF;
END_REGION

REGION Network 10 (SCL): Re_Home
   IF #"RW Done" = TRUE & #Re_home = TRUE & #"Process".mobusMaster.Busy = FALSE THEN
       IF #"Process".Step_W = 1 THEN
           #"Process".Step_W := 2;
           #"Process".Step := 1;
           #"Process".SinggleData[0] := -100;
       ELSIF #"Process".Step_W = 2 THEN
           #"Process".Step_W := 3;
           #"Process".Step := 1;
           #"Process".SinggleData[0] := 80;
           #Process.SinggleData[1] := 0;
       ELSIF #"Process".Step_W = 3 THEN
           #"Process".Step_W := 5;
           #"Process".Step := 1;
           #"Process".SinggleData[0] := 31;
           ;
       ELSIF #"Process".Step_W = 5 THEN
           #"Process".Step_W := 0;
           #"Process".Step := 0;
           #"Enable_Write" := FALSE;
           #Re_home := FALSE;
           #Re_home_Excuting := TRUE;
           #Write_Full_Done := TRUE;
           // <Enable read to read Alarm>
           // 
           // Statement
           // 
           //<End>
           ;
       END_IF;
       ;
   END_IF;
END_REGION

REGION Network 11 (SCL): MOVE HOME
   IF #"RW Done" = TRUE & #Move_Home = TRUE & #"Process".mobusMaster.Busy = FALSE THEN
       IF #"Process".Step_W = 1 THEN
           #"Process".Step_W := 2;
           #"Process".Step := 1;
           #"Process".SinggleData[0] := -100;
       ELSIF #"Process".Step_W = 2 THEN
           #"Process".Step_W := 3;
           #"Process".Step := 1;
           #"Process".SinggleData[0] := #Home_Speed;
           #Process.SinggleData[1] := 0;
       ELSIF #"Process".Step_W = 3 THEN
           #"Process".Step_W := 5;
           #"Process".Step := 1;
           #"Process".SinggleData[0] := 31;
           ;
       ELSIF #"Process".Step_W = 5 THEN
           #"Process".Step_W := 0;
           #"Process".Step := 0;
           #"Enable_Write" := FALSE;
           #Move_Home := FALSE;
           #Jog_FW_Home_Excuting := TRUE;
           #Write_Full_Done := TRUE;
           // <Enable read to read Alarm>
           // 
           // Statement
           // 
           //<End>
           ;
       END_IF;
       ;
   END_IF;
END_REGION

REGION Network 12 (SCL): Reset Fault
   IF #"RW Done" = TRUE &#"Reset_fault" = TRUE &#"Process".mobusMaster.Busy = FALSE THEN
       ;
       IF #"Process".Step_W = 1 THEN
           #"Process".Step_W := 0;
           #"Process".Step := 0;
           #"Reset_fault" := FALSE;
           #Enable_Write := FALSE;
           #Write_Full_Done := TRUE;
           ;
       END_IF;
   END_IF;
END_REGION

REGION Network 13 (SCL): Reset_servo
   IF #"RW Done" = TRUE & #Reset_Servo = TRUE & #"Process".mobusMaster.Busy = FALSE THEN
       ;
       IF #"Process".Step_W = 3 THEN
           #"Process".Step_W := 0;
           #"Process".Step := 0;
           #Reset_Servo := FALSE;
           #Write_Full_Done := TRUE;
           #Enable_Write := FALSE;
           ;
       END_IF;
   END_IF;
END_REGION

REGION Network 14 (SCL): HOMING
   IF #"RW Done" = TRUE &#"HOME" = TRUE &#"Process".mobusMaster.Busy = FALSE THEN
       IF #"Process".Step_W = 1 THEN
           #"Process".Step_W := 2;
           #"Process".Step := 1;
           #"Process".SinggleData[0] := 6;
       ELSIF #"Process".Step_W = 2 THEN
           #"Process".Step_W := 3;
           #"Process".Step := 1;
           #"Process".SinggleData[0] := 150;
       ELSIF #"Process".Step_W = 3 THEN
           #"Process".Step_W := 6;
           #"Process".Step := 1;
           #"Process".SinggleData[0] := 35;
           ; 
       ELSIF #"Process".Step_W = 6 THEN
           #"Process".Step_W := 5;
           #"Process".Step := 1;
           #"Process".SinggleData[0] := 31;
           ;
       ELSIF #"Process".Step_W = 5 THEN
           #"Process".Step_W := 0;
           #"Process".Step := 0;
           #"HOME" := FALSE;
           #"Enable_Write" := FALSE;
           #Write_Full_Done := TRUE;
           ;
       END_IF;
       ;
   END_IF;
END_REGION

REGION Network 15 (SCL): JOG+
   IF #"RW Done" = TRUE &#"Jog+" = TRUE &#"Process".mobusMaster.Busy = FALSE THEN
       IF #"Process".Step_W = 1 THEN
           #"Process".Step_W := 2;
           #"Process".Step := 1;
           #"Process".SinggleData[0] := -100;
       ELSIF #"Process".Step_W = 2 THEN
           #"Process".Step_W := 3;
           #"Process".Step := 1;
           #"Process".SinggleData[0] := #Jog_Speed;
           #Process.SinggleData[1] := 0;
       ELSIF #"Process".Step_W = 3 THEN
           #"Process".Step_W := 5;
           #"Process".Step := 1;
           #"Process".SinggleData[0] := 31;
           ;
       ELSIF #"Process".Step_W = 5 THEN
           #"Process".Step_W := 0;
           #"Process".Step := 0;
           #"DisJog+" := TRUE;
           #"Enable_Write" := FALSE;
           #Write_Full_Done := TRUE;
           ;
       END_IF;
       ;
   END_IF;
   IF #"RW Done" = TRUE & #Process.mobusMaster.Busy = FALSE & #"DisJog+" = TRUE & #"Jog+" = FALSE THEN
       ;
       IF #Process.Step_W = 1 THEN
           ;
           #Process.Step_W := 0;
           #Process.Step := 0;
           #"Enable_Write" := FALSE;
           #Write_Full_Done := TRUE;
           #"DisJog+" := FALSE;
       END_IF;
   END_IF;
END_REGION

REGION Network 16 (SCL): JOG-
   IF #"RW Done" = TRUE &#"Jog-" = TRUE &#"Process".mobusMaster.Busy = FALSE &#"DisJog-" = TRUE THEN
       IF #"Process".Step_W = 1 THEN
           #"Process".Step_W := 2;
           #"Process".Step := 1;
           #"Process".SinggleData[0] := -100;
       ELSIF #"Process".Step_W = 2 THEN
           #"Process".Step_W := 3;
           #"Process".Step := 1;
           #"Process".SinggleData[0] := #Jog_Speed;
           #Process.SinggleData[1] := 0;
       ELSIF #"Process".Step_W = 3 THEN
           #"Process".Step_W := 5;
           #"Process".Step := 1;
           #"Process".SinggleData[0] := 63;
           ;
       ELSIF #"Process".Step_W = 5 THEN
           #"Process".Step_W := 0;
           #"Process".Step := 0;
           #"DisJog-" := TRUE;
           #"Enable_Write" := FALSE;
           #Write_Full_Done := TRUE;
           ;
       END_IF;
       ;
   END_IF;
   IF #"RW Done" = TRUE & #Process.mobusMaster.Busy = FALSE & #"DisJog-" = TRUE & #"Jog-" = FALSE THEN
       ;
       IF #Process.Step_W = 1 THEN
           ;
           #Process.Step_W := 0;
           #Process.Step := 0;
           #"Enable_Write" := FALSE;
           #Write_Full_Done := TRUE;
           #"DisJog-" := FALSE;
       END_IF;
   END_IF;
END_REGION

REGION Network 17 (SCL): MOVE POINT
   IF #"RW Done" = TRUE &#"Move_point" = TRUE &#"Process".mobusMaster.Busy = FALSE THEN
       ;
       IF #"Process".Step_W = 1 THEN
           ;
           #"Process".Step_W := 2;
           #"Process".SinggleData[0] := -101;
           #"Process".Step := 1;
       ELSIF #"Process".Step_W = 2 THEN
           #"Process".Step_W := 4;
           #"Process".SinggleData[0] := #Select_Point;
           #"Process".Step := 1;
       ELSIF #"Process".Step_W = 4 THEN
           #"Process".Step_W := 5;
           #"Process".SinggleData[0] := 31;
           #"Process".Step := 1;
       ELSIF #"Process".Step_W = 5 THEN
           #"Process".Step_W := 0;
           #"Process".Step := 0;
           #"Move_point" := FALSE;
           #"Enable_Write" := FALSE;
           //#"Enable Read" := TRUE;
           #Write_Full_Done := TRUE;
       END_IF;
   END_IF;
END_REGION

REGION Network 18 (SCL): Set_point
   IF #"Set_point" = TRUE &#"Process".mobusMaster.Busy = FALSE &#"RW Done" = TRUE THEN
       ;
       IF #"Process".Step_W > 10 THEN
           ;
           #"Process".Step_W := 0;
           #"Process".Step := 0;
           #"Set_point" := FALSE;
           #"Enable_Write" := FALSE;
           #"Enable Read" := TRUE;
           #Write_Full_Done := TRUE;
       END_IF;
   END_IF;
END_REGION

REGION Network 19: Output Pin
   RUNG wire#powerrail
      Contact( #Enable_block )
      Contact( #Process.mobusMaster.Req )
      Coil( #Req )
   END_RUNG
   RUNG wire#powerrail
      Contact( #Read_Full_Done )
      Contact( #Write_Full_Done )
      Coil( #All_Done )
   END_RUNG
   // the same network as SCL:
   #Req := #Enable_block AND #Process.mobusMaster.Req;
   #All_Done := #Read_Full_Done AND #Write_Full_Done;
END_REGION
END_FUNCTION_BLOCK

FUNCTION_BLOCK "Inventer_Control"   // FB9, LAD
{ S7_Optimized_Access := 'TRUE' }
VERSION : 0.1
   VAR_INPUT
      Busy : Bool;
      Done : Bool;
      Error : Bool;
      Status : Word;
      Enable_block : Bool;
   END_VAR
   VAR_OUTPUT
      Req : Bool;
      Mb_ID : UInt;
      DataLen : UInt := 1;
      DataAddr : UDInt;
      Mode : UInt;
   END_VAR
   VAR_IN_OUT
      Ptr : Array[0..8] of Int;
   END_VAR
   VAR
      Process : "Process";
      ID : Int := 3;
      Data_Ptr : Array[0..8] of Int;
      Data_Ptr_Received : Array[0..8] of Int;
      Data_Ptr_Send : Array[0..8] of Int;
   END_VAR
   VAR RETAIN
      Frequency : Real := 50.0;
   END_VAR
   VAR
      Accel_time : Real := 0.5;
      Decel_time : Real := 0.5;
      Max_Frequency : Real := 150.0;
      cvt_Freq : Int := 1;
      cvt_MaxFreq : Int := 1;
      cvt_Accel : Int := 1;
      cvt_Decel : Int := 1;
      "Jog-" : Bool;
      "Jog+" : Bool;
      "RW Done" : Bool;
      Enable_Write : Bool;
      "DisJog-" : Bool;
      "DisJog+" : Bool;
      "Enable Read" : Bool;
      All_Done : Bool := true;
      Write_Full_Done : Bool := true;
      Read_Full_Done : Bool := true;
      delay_rs : Time := T#400ms;
      Run_FW : Bool;
      Run_BW : Bool;
      Stop_Jog : Bool;
      Stop_Run : Bool;
      Reset_fault : Bool;
      Set_Freqency : Bool;
      Set_MaxFreq : Bool;
      Set_Accel_Decc : Bool;
      Data_Freqency : Int;
      Data_Accel_Time : Int;
      Data_Deccel_Time : Int;
      Data_Status : Int := 4;   // 1: fw running, 2 bw running, 3: stop, 4: stop, POFF state
      Data_Current : Int;
      Stop_FW : Bool;
      Stop_BW : Bool;
   END_VAR
   VAR_TEMP
      temp : Real;
      temp1 : Real;
      temp2 : Real;
      temp3 : Real;
   END_VAR
   VAR_TEMP   // added for the SCL form of the ladder/FBD networks
      _w1 : Bool;
      _w2 : Bool;
      _w3 : Bool;
      _w4 : Bool;
      _w5 : Bool;
      _w6 : Bool;
      _w7 : Bool;
      _w8 : Bool;
      _w9 : Bool;
      _w10 : Bool;
      _w11 : Bool;
      _w12 : Bool;
      _w13 : Bool;
   END_VAR
BEGIN

REGION Network 1 (SCL)
   IF #Process.Step = 1 THEN
       ;
       #Process.mobusMaster.Mode := 2;
       #Mode := #Process.mobusMaster.Mode;
       #Process.mobusMaster.MbAddress := #ID;
       #Mb_ID := INT_TO_UINT(#Process.mobusMaster.MbAddress);
       IF #Process.Step_W = 1 THEN
           ;
           //Thanh ghi Command
           // 1: fw run
           // 2: rev un
           // 3 fw jog
           // 4 rev jog
           // 5 stop run
           // 6 EMG stop
           // 7 reset fault
           // 8 jog stop
           #Process.mobusMaster.DataAddr := 48193;
           #DataAddr := #Process.mobusMaster.DataAddr;
       ELSIF #Process.Step_W = 2 THEN
           ;
           //Thanh GHi Tần số
           #Process.mobusMaster.DataAddr := 48194;
           #DataAddr := #Process.mobusMaster.DataAddr;
       ELSIF #Process.Step_W = 3 THEN
           ;
           // max frequency
           #Process.mobusMaster.DataAddr := 40004;
           #DataAddr := #Process.mobusMaster.DataAddr;
       ELSIF #Process.Step_W = 4 THEN
           ;
           //Accelerate
           #Process.mobusMaster.DataAddr := 40012;
           #DataAddr := #Process.mobusMaster.DataAddr;

       END_IF;

       #Data_Ptr_Send := #Process.SinggleData;
       IF #Process.Step_W = 4 THEN
           ;
           #Process.mobusMaster.DataLen := 2;
           #DataLen := #Process.mobusMaster.DataLen;
       ELSE
           ;
           #Process.mobusMaster.DataLen := 1;
           #DataLen := #Process.mobusMaster.DataLen;
       END_IF;


       #Data_Ptr := #Data_Ptr_Send;
       #Ptr := #Data_Ptr;

       #Process.mobusMaster.Req := TRUE;

       IF #Process.mobusMaster.Busy THEN
           ;
           #Process.Step := 2;
       END_IF;

   ELSIF #Process.Step = 2 THEN
       ;
       IF #Process.mobusMaster.Done THEN
           ;
           #Process.mobusMaster.Req := FALSE;
           #Process.Step := 5;
       END_IF;
   ELSIF #Process.Step = 3 THEN
       ;
       #Process.mobusMaster.Mode := 0;
       #Mode := #Process.mobusMaster.Mode;
       #Process.mobusMaster.MbAddress := #ID;
       #Mb_ID := INT_TO_UINT(#Process.mobusMaster.MbAddress);
       IF #Process.Step_R = 1 THEN
           ;
           //read frequency
           #Process.mobusMaster.DataAddr := 48194;
           #DataAddr := #Process.mobusMaster.DataAddr;
           #Process.mobusMaster.DataLen := 1;
           #DataLen := #Process.mobusMaster.DataLen;
       ELSIF #Process.Step_R = 2 THEN
           ;
           // read status
           #Process.mobusMaster.DataAddr := 48449;
           #DataAddr := #Process.mobusMaster.DataAddr;
           #Process.mobusMaster.DataLen := 1;
           #DataLen := #Process.mobusMaster.DataLen;
       ELSIF #Process.Step_R = 3 THEN
           ;
           //read accel
           #Process.mobusMaster.DataAddr := 40012;
           #DataAddr := #Process.mobusMaster.DataAddr;
           #Process.mobusMaster.DataLen := 2;
           #DataLen := #Process.mobusMaster.DataLen;
       ELSIF #Process.Step_R = 4 THEN
           ;
           //read Current
           #Process.mobusMaster.DataAddr := 412293;
           #DataAddr := #Process.mobusMaster.DataAddr;
           #Process.mobusMaster.DataLen := 1;
           #DataLen := #Process.mobusMaster.DataLen;
       END_IF;

       #Process.mobusMaster.Req := TRUE;
       IF #Process.mobusMaster.Busy = TRUE THEN
           ;
           #Process.Step := 4;
       END_IF;
   ELSIF #Process.Step = 4 & #Process.mobusMaster.Done = TRUE THEN
       ;
       #Process.mobusMaster.Req := FALSE;

       IF #Process.Step_R = 1  THEN
           ;
           #Data_Ptr_Received := #Ptr;
           #Data_Freqency := #Data_Ptr_Received[0];

       ELSIF #Process.Step_R = 2 THEN
           ;
           //Status
           #Data_Ptr_Received := #Ptr;
           #Data_Status := #Data_Ptr_Received[0];

       ELSIF #Process.Step_R = 3 THEN
           ;
           // accel
           #Data_Ptr_Received := #Ptr;
           #Data_Accel_Time := #Data_Ptr_Received[0];
           //decel
           #Data_Deccel_Time := #Data_Ptr_Received[1];
       ELSIF #Process.Step_R = 4 THEN
           ;
           //Current
           #Data_Ptr_Received := #Ptr;
           #Data_Current := #Data_Ptr_Received[0];
       END_IF;
       #Process.Step := 5;
       END_IF;
END_REGION

REGION Network 2: Input pin
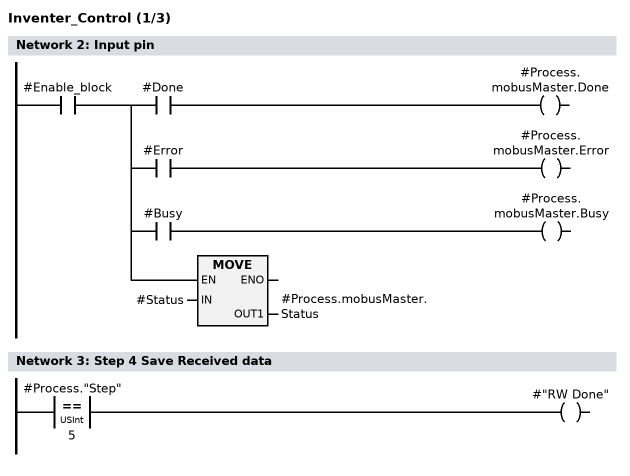
   RUNG wire#powerrail
      Contact( #Enable_block )
      wire#w1
      Contact( #Done )
      Coil( #Process.mobusMaster.Done )
   END_RUNG
   RUNG wire#w1
      Contact( #Error )
      Coil( #Process.mobusMaster.Error )
   END_RUNG
   RUNG wire#w1
      Contact( #Busy )
      Coil( #Process.mobusMaster.Busy )
   END_RUNG
   RUNG wire#w1
      Move(in := #Status, out1 => #Process.mobusMaster.Status)
   END_RUNG
   // the same network as SCL:
   #Process.mobusMaster.Done := #Enable_block AND #Done;
   #Process.mobusMaster.Error := #Enable_block AND #Error;
   #Process.mobusMaster.Busy := #Enable_block AND #Busy;
   IF #Enable_block THEN #Process.mobusMaster.Status := #Status; END_IF;
END_REGION

REGION Network 3: Step 4 Save Received data
   RUNG wire#powerrail
      { S7_Templates := "SrcType := USInt" } EQ_Contact(in1 := #Process."Step", in2 := 5)
      Coil( #"RW Done" )
   END_RUNG
   // the same network as SCL:
   #"RW Done" := #Process."Step" = 5;
END_REGION

REGION Network 4: Excute Command
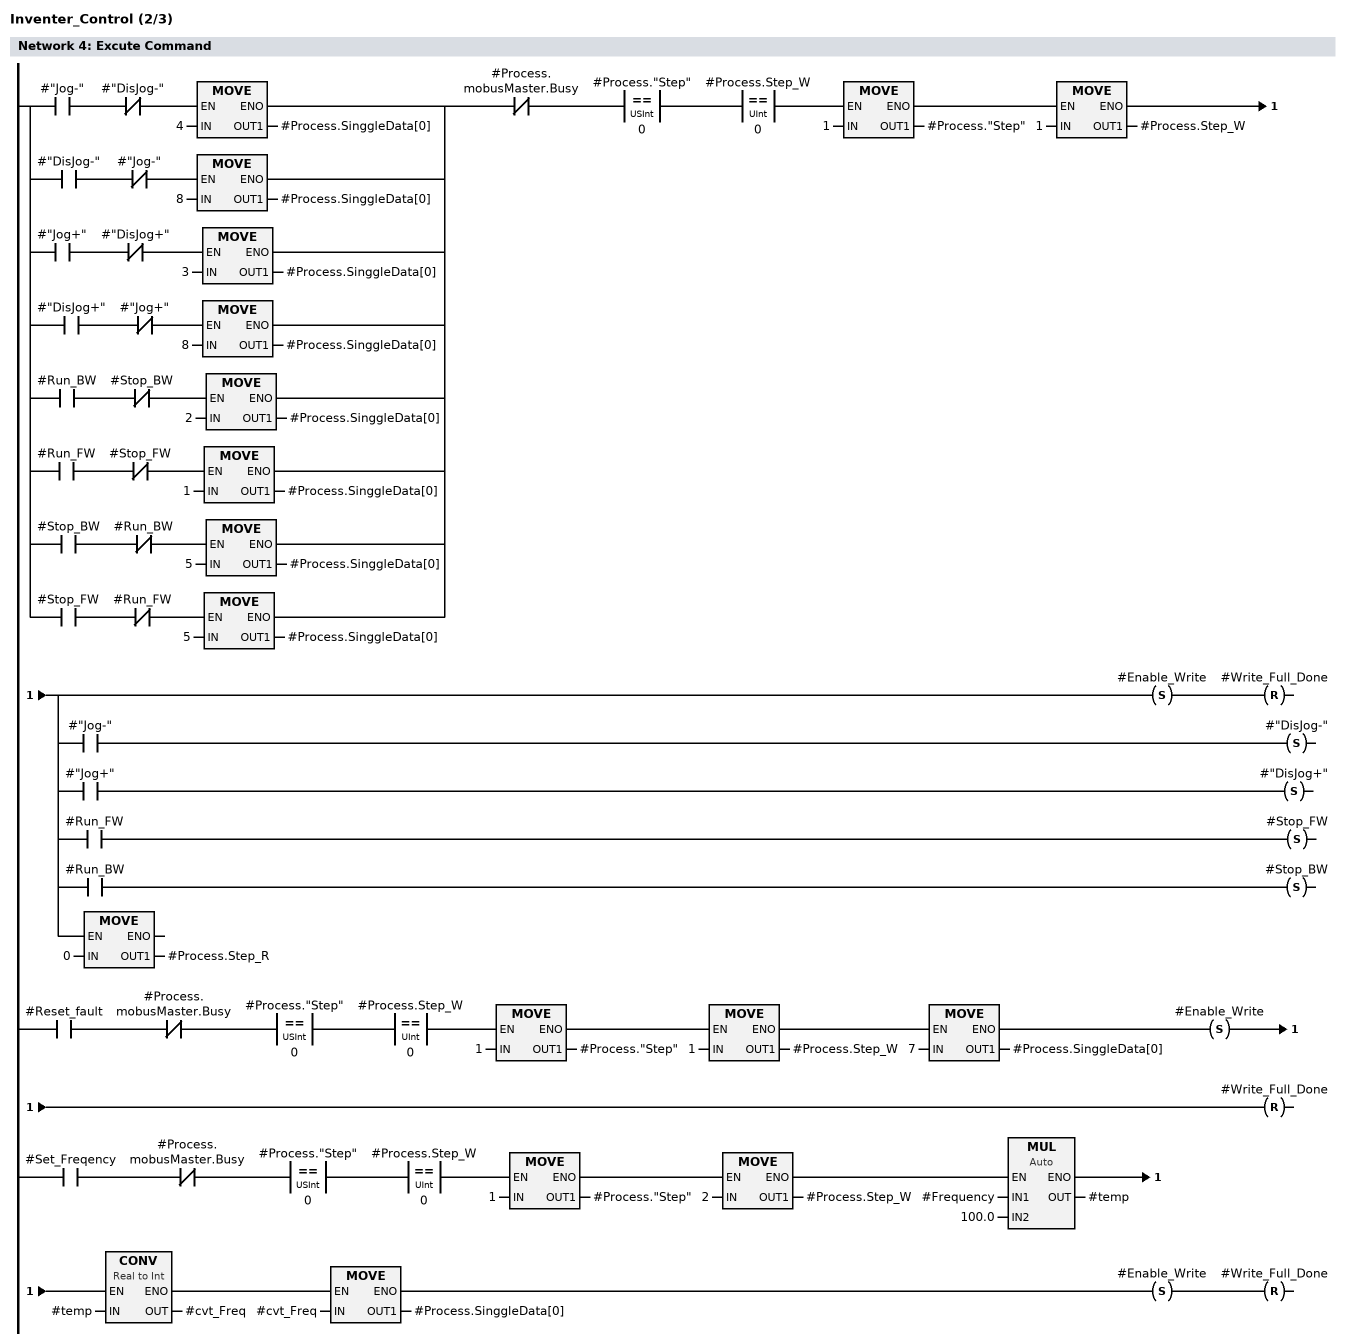
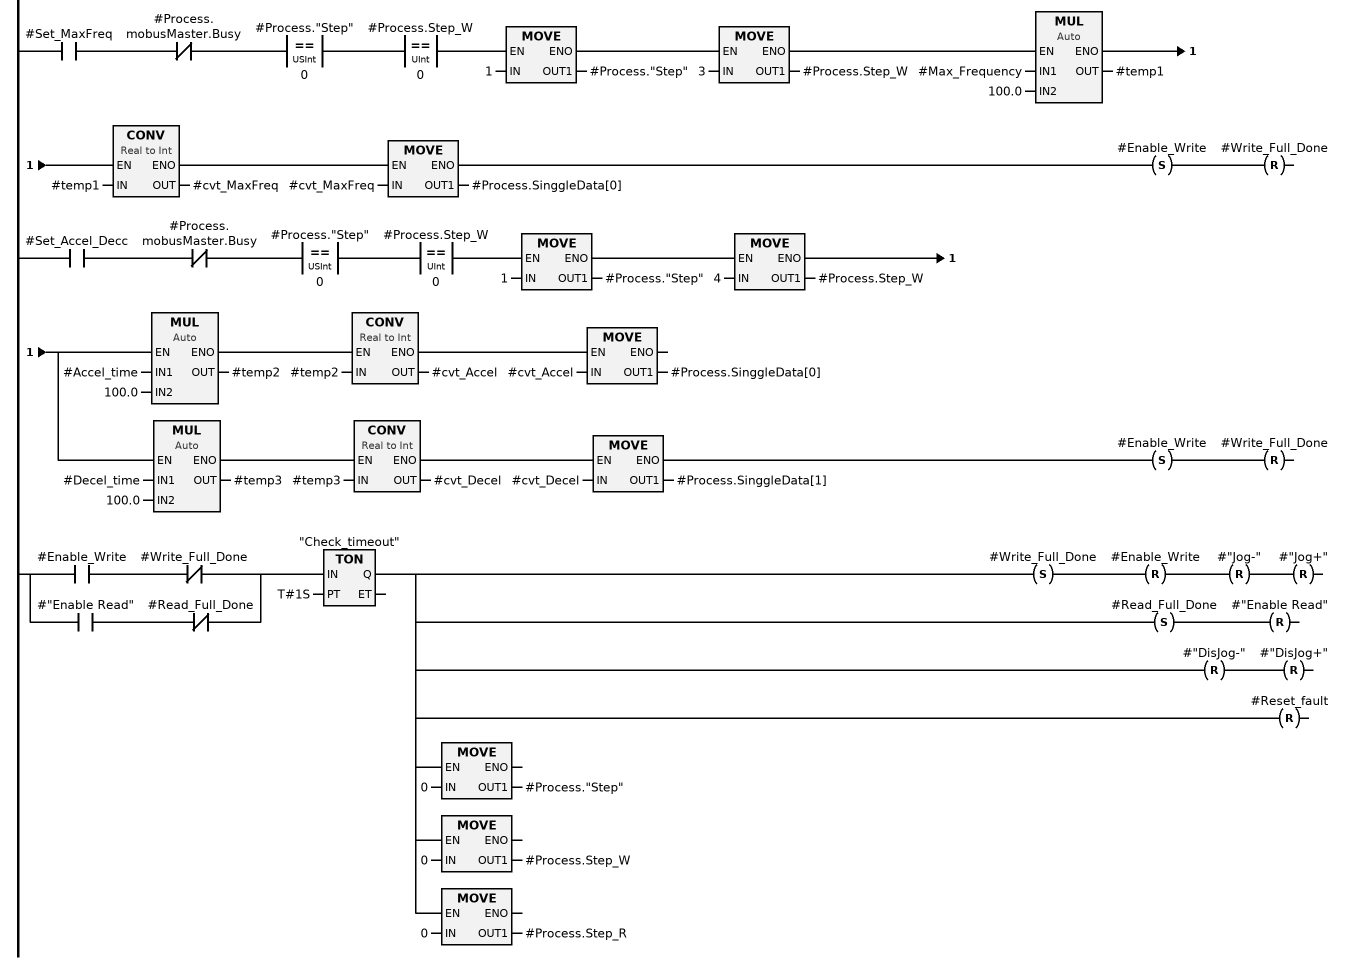
   // ENO of a box is taken as its EN; it also drops when the box reports an error
   #_w1 := #"Jog-" AND NOT #"DisJog-";
   IF #_w1 THEN #Process.SinggleData[0] := 4; END_IF;
   #_w2 := #"DisJog-" AND NOT #"Jog-";
   IF #_w2 THEN #Process.SinggleData[0] := 8; END_IF;
   #_w3 := #"Jog+" AND NOT #"DisJog+";
   IF #_w3 THEN #Process.SinggleData[0] := 3; END_IF;
   #_w4 := #"DisJog+" AND NOT #"Jog+";
   IF #_w4 THEN #Process.SinggleData[0] := 8; END_IF;
   #_w5 := #Run_BW AND NOT #Stop_BW;
   IF #_w5 THEN #Process.SinggleData[0] := 2; END_IF;
   #_w6 := #Run_FW AND NOT #Stop_FW;
   IF #_w6 THEN #Process.SinggleData[0] := 1; END_IF;
   #_w7 := #Stop_BW AND NOT #Run_BW;
   IF #_w7 THEN #Process.SinggleData[0] := 5; END_IF;
   #_w8 := #Stop_FW AND NOT #Run_FW;
   IF #_w8 THEN #Process.SinggleData[0] := 5; END_IF;
   #_w9 := (#_w1 OR #_w2 OR #_w3 OR #_w4 OR #_w5 OR #_w6 OR #_w7 OR #_w8) AND NOT #Process.mobusMaster.Busy AND (#Process."Step" = 0) AND (#Process.Step_W = 0);
   IF #_w9 THEN
       #Process."Step" := 1;
       #Process.Step_W := 1;
       #Enable_Write := TRUE;
       #Write_Full_Done := FALSE;
   END_IF;
   IF #_w9 AND #"Jog-" THEN #"DisJog-" := TRUE; END_IF;
   IF #_w9 AND #"Jog+" THEN #"DisJog+" := TRUE; END_IF;
   IF #_w9 AND #Run_FW THEN #Stop_FW := TRUE; END_IF;
   IF #_w9 AND #Run_BW THEN #Stop_BW := TRUE; END_IF;
   IF #_w9 THEN #Process.Step_R := 0; END_IF;
   #_w10 := #Reset_fault AND NOT #Process.mobusMaster.Busy AND (#Process."Step" = 0) AND (#Process.Step_W = 0);
   IF #_w10 THEN
       #Process."Step" := 1;
       #Process.Step_W := 1;
       #Process.SinggleData[0] := 7;
       #Enable_Write := TRUE;
       #Write_Full_Done := FALSE;
   END_IF;
   #_w11 := #Set_Freqency AND NOT #Process.mobusMaster.Busy AND (#Process."Step" = 0) AND (#Process.Step_W = 0);
   IF #_w11 THEN
       #Process."Step" := 1;
       #Process.Step_W := 2;
       #temp := #Frequency * 100.0;
       #cvt_Freq := REAL_TO_INT(#temp);
       #Process.SinggleData[0] := #cvt_Freq;
       #Enable_Write := TRUE;
       #Write_Full_Done := FALSE;
   END_IF;
   #_w12 := #Set_MaxFreq AND NOT #Process.mobusMaster.Busy AND (#Process."Step" = 0) AND (#Process.Step_W = 0);
   IF #_w12 THEN
       #Process."Step" := 1;
       #Process.Step_W := 3;
       #temp1 := #Max_Frequency * 100.0;
       #cvt_MaxFreq := REAL_TO_INT(#temp1);
       #Process.SinggleData[0] := #cvt_MaxFreq;
       #Enable_Write := TRUE;
       #Write_Full_Done := FALSE;
   END_IF;
   #_w13 := #Set_Accel_Decc AND NOT #Process.mobusMaster.Busy AND (#Process."Step" = 0) AND (#Process.Step_W = 0);
   IF #_w13 THEN
       #Process."Step" := 1;
       #Process.Step_W := 4;
       #temp2 := #Accel_time * 100.0;
       #cvt_Accel := REAL_TO_INT(#temp2);
       #Process.SinggleData[0] := #cvt_Accel;
       #temp3 := #Decel_time * 100.0;
       #cvt_Decel := REAL_TO_INT(#temp3);
       #Process.SinggleData[1] := #cvt_Decel;
       #Enable_Write := TRUE;
       #Write_Full_Done := FALSE;
   END_IF;
   "Check_timeout".TON(IN := (#Enable_Write AND NOT #Write_Full_Done) OR (#"Enable Read" AND NOT #Read_Full_Done),
                       PT := T#1S);
   IF "Check_timeout".Q THEN
       #Write_Full_Done := TRUE;
       #Enable_Write := FALSE;
       #"Jog-" := FALSE;
       #"Jog+" := FALSE;
       #Read_Full_Done := TRUE;
       #"Enable Read" := FALSE;
       #"DisJog-" := FALSE;
       #"DisJog+" := FALSE;
       #Reset_fault := FALSE;
       #Process."Step" := 0;
       #Process.Step_W := 0;
       #Process.Step_R := 0;
   END_IF;
END_REGION

REGION Network 5: Read Control
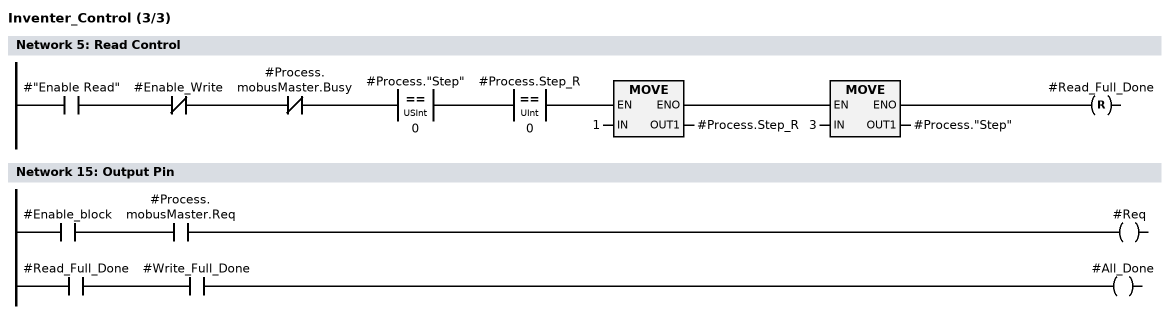
   RUNG wire#powerrail
      Contact( #"Enable Read" )
      I_Contact( #Enable_Write )
      I_Contact( #Process.mobusMaster.Busy )
      { S7_Templates := "SrcType := USInt" } EQ_Contact(in1 := #Process."Step", in2 := 0)
      { S7_Templates := "SrcType := UInt" } EQ_Contact(in1 := #Process.Step_R, in2 := 0)
      Move(in := 1, out1 => #Process.Step_R)
      Move(in := 3, out1 => #Process."Step")
      R_Coil( #Read_Full_Done )
   END_RUNG
   // the same network as SCL:
   #_w1 := #"Enable Read" AND NOT #Enable_Write AND NOT #Process.mobusMaster.Busy AND (#Process."Step" = 0) AND (#Process.Step_R = 0);
   IF #_w1 THEN
       #Process.Step_R := 1;
       #Process."Step" := 3;
       #Read_Full_Done := FALSE;
   END_IF;
END_REGION

REGION Network 6 (SCL): Read Process
   IF #"Enable Read"= TRUE & #"Process".mobusMaster.Busy = FALSE & #"RW Done"= TRUE & #"Enable_Write" = FALSE THEN
       ;
       IF #"Process".Step_R = 1 THEN
           #"Process".Step_R := 2;
           #"Process".Step := 3;
       ELSIF #"Process".Step_R = 2 THEN
           #"Process".Step_R := 3;
           #"Process".Step := 3;
       ELSIF #"Process".Step_R = 3 THEN
           #"Process".Step_R := 4;
           #"Process".Step := 3;
           // Done read Signed
       ELSIF #Process.Step_R = 4 THEN
           ;
           #Process.Step := 0;
           #Process.Step_R := 0;
           #"Enable Read" := FALSE;
           #Read_Full_Done := TRUE;

       END_IF;
   ELSIF #"Process".mobusMaster.Busy = FALSE &#"Process".Step_R <> 0 &#"RW Done" = TRUE &#"Enable_Write" = TRUE THEN
       ;
       #"Process".Step_R := 0;
       #"Process".Step := 0;
       #Read_Full_Done := TRUE;
   ELSIF #"Process".mobusMaster.Busy = FALSE &#"Process".Step_R <> 0 &#"Enable_Write" = FALSE &#"Enable Read" = FALSE &#"Process".Step <> 0 THEN
       ;
       #"Process".Step_R := 0;
       #"Process".Step := 0;
       #Read_Full_Done := TRUE;
   END_IF;
END_REGION

REGION Network 7 (SCL): Reset Fault
   IF #"RW Done" = TRUE &#"Reset_fault" = TRUE &#"Process".mobusMaster.Busy = FALSE THEN
       ;
       IF #"Process".Step_W = 1 THEN
           #"Process".Step_W := 0;
           #"Process".Step := 0;
           #"Reset_fault" := FALSE;
           #Enable_Write := FALSE;
           #Write_Full_Done := TRUE;
           ;
       END_IF;
   END_IF;
END_REGION

REGION Network 8 (SCL): JOG+
   IF #"RW Done" = TRUE &#"Jog+" = TRUE &#"Process".mobusMaster.Busy = FALSE THEN
       IF #"Process".Step_W = 1 THEN
           #"Process".Step_W := 0;
           #"Process".Step := 0;
           #"DisJog+" := TRUE;
           #"Enable_Write" := FALSE;
           #Write_Full_Done := TRUE;
           ;
       END_IF;
       ;
   END_IF;
   IF #"RW Done" = TRUE & #Process.mobusMaster.Busy = FALSE & #"DisJog+" = TRUE & #"Jog+" = FALSE THEN
       ;
       IF #Process.Step_W = 1 THEN
           ;
           #Process.Step_W := 0;
           #Process.Step := 0;
           #"Enable_Write" := FALSE;
           #Write_Full_Done := TRUE;
           #"DisJog+" := FALSE;
       END_IF;
   END_IF;
END_REGION

REGION Network 9 (SCL): JOG-
   IF #"RW Done" = TRUE &#"Jog-" = TRUE &#"Process".mobusMaster.Busy = FALSE &#"DisJog-" = TRUE THEN
       IF #"Process".Step_W = 1 THEN
           #"Process".Step_W := 0;
           #"Process".Step := 0;
           #"DisJog-" := TRUE;
           #"Enable_Write" := FALSE;
           #Write_Full_Done := TRUE;
           ;
       END_IF;
       ;
   END_IF;
   IF #"RW Done" = TRUE & #Process.mobusMaster.Busy = FALSE & #"DisJog-" = TRUE & #"Jog-" = FALSE THEN
       ;
       IF #Process.Step_W = 1 THEN
           ;
           #Process.Step_W := 0;
           #Process.Step := 0;
           #"Enable_Write" := FALSE;
           #Write_Full_Done := TRUE;
           #"DisJog-" := FALSE;
       END_IF;
   END_IF;
END_REGION

REGION Network 10 (SCL): RUN BW
   IF #"RW Done" = TRUE & #Run_BW = TRUE & #"Process".mobusMaster.Busy = FALSE THEN
       IF #"Process".Step_W = 1 THEN
           #"Process".Step_W := 0;
           #"Process".Step := 0;
           #Stop_BW := TRUE;
           #"Enable_Write" := FALSE;
           #Write_Full_Done := TRUE;
           ;
       END_IF;
       ;
   END_IF;
   IF #"RW Done" = TRUE & #Process.mobusMaster.Busy = FALSE & #Stop_BW = TRUE & #Run_BW = FALSE THEN
       ;
       IF #Process.Step_W = 1 THEN
           ;
           #Process.Step_W := 0;
           #Process.Step := 0;
           #"Enable_Write" := FALSE;
           #Write_Full_Done := TRUE;
           #Stop_BW := FALSE;
       END_IF;
   END_IF;
END_REGION

REGION Network 11 (SCL): RUN FW
   IF #"RW Done" = TRUE & #Run_FW = TRUE & #"Process".mobusMaster.Busy = FALSE THEN
       IF #"Process".Step_W = 1 THEN
           #"Process".Step_W := 0;
           #"Process".Step := 0;
           #Stop_FW := TRUE;
           #"Enable_Write" := FALSE;
           #Write_Full_Done := TRUE;
           ;
       END_IF;
       ;
   END_IF;
   IF #"RW Done" = TRUE & #Process.mobusMaster.Busy = FALSE & #Stop_FW = TRUE & #Run_FW = FALSE THEN
       ;
       IF #Process.Step_W = 1 THEN
           ;
           #Process.Step_W := 0;
           #Process.Step := 0;
           #"Enable_Write" := FALSE;
           #Write_Full_Done := TRUE;
           #Stop_FW := FALSE;
       END_IF;
   END_IF;
END_REGION

REGION Network 12 (SCL): Set_freqency
   IF #"RW Done" = TRUE & #Set_Freqency = TRUE & #"Process".mobusMaster.Busy = FALSE THEN
       ;
       IF #"Process".Step_W = 2 THEN
           #"Process".Step_W := 0;
           #"Process".Step := 0;
           #Set_Freqency := FALSE;
           #Enable_Write := FALSE;
           #Write_Full_Done := TRUE;
           ;
       END_IF;
   END_IF;
END_REGION

REGION Network 13 (SCL): Set Max Freq
   IF #"RW Done" = TRUE & #Set_MaxFreq = TRUE & #"Process".mobusMaster.Busy = FALSE THEN
       ;
       IF #"Process".Step_W = 3 THEN
           #"Process".Step_W := 0;
           #"Process".Step := 0;
           #Set_MaxFreq := FALSE;
           #Enable_Write := FALSE;
           #Write_Full_Done := TRUE;
           ;
       END_IF;
   END_IF;
END_REGION

REGION Network 14 (SCL): Set Accel
   IF #"RW Done" = TRUE & #Set_Accel_Decc = TRUE & #"Process".mobusMaster.Busy = FALSE THEN
       ;
       IF #"Process".Step_W = 4 THEN
           #"Process".Step_W := 0;
           #"Process".Step := 0;
           #Process.SinggleData[1] := 0;
           #Set_Accel_Decc := FALSE;
           #Enable_Write := FALSE;
           #Write_Full_Done := TRUE;
           ;
       END_IF;
   END_IF;
END_REGION

REGION Network 15: Output Pin
   RUNG wire#powerrail
      Contact( #Enable_block )
      Contact( #Process.mobusMaster.Req )
      Coil( #Req )
   END_RUNG
   RUNG wire#powerrail
      Contact( #Read_Full_Done )
      Contact( #Write_Full_Done )
      Coil( #All_Done )
   END_RUNG
   // the same network as SCL:
   #Req := #Enable_block AND #Process.mobusMaster.Req;
   #All_Done := #Read_Full_Done AND #Write_Full_Done;
END_REGION
END_FUNCTION_BLOCK

FUNCTION "SHIFT_RIGHT_DATA_AREA1_3" : Void   // FC1, SCL
{ S7_Optimized_Access := 'TRUE' }
VERSION : 0.1
   VAR_TEMP
      Check_Has_Barcode : Bool;
   END_VAR
BEGIN
   // Area 3

